LIN {X -0.056,Y -514.496,Z 256.006,A 0.000,B 0.000,C 90.000,E1 217.076} C_DIS
LIN {X -0.191,Y -508.629,Z 255.995,A 0.000,B 0.000,C 90.000,E1 215.025} C_DIS
LIN {X 0.078,Y -502.743,Z 255.983,A 0.000,B 0.000,C 90.000,E1 212.911} C_DIS
LIN {X -0.204,Y -496.416,Z 255.970,A 0.000,B 0.000,C 90.000,E1 210.541} C_DIS
LIN {X 0.173,Y -489.660,Z 255.954,A 0.000,B 0.000,C 90.000,E1 207.769} C_DIS
LIN {X -0.155,Y -484.810,Z 255.943,A 0.000,B 0.000,C 90.000,E1 205.668} C_DIS
LIN {X -0.161,Y -481.730,Z 255.934,A 0.000,B 0.000,C 90.000,E1 204.131} C_DIS
LIN {X -0.246,Y -475.770,Z 255.917,A 0.000,B 0.000,C 90.000,E1 201.046} C_DIS
LIN {X -0.152,Y -472.029,Z 255.905,A 0.000,B 0.000,C 90.000,E1 198.852} C_DIS
LIN {X -0.121,Y -469.175,Z 255.894,A 0.000,B 0.000,C 90.000,E1 196.968} C_DIS
LIN {X -0.013,Y -465.218,Z 255.878,A 0.000,B 0.000,C 90.000,E1 194.120} C_DIS
LIN {X -0.052,Y -462.080,Z 255.864,A 0.000,B 0.000,C 90.000,E1 191.591} C_DIS
LIN {X -0.160,Y -459.448,Z 255.852,A 0.000,B 0.000,C 90.000,E1 189.378} C_DIS
LIN {X 0.145,Y -456.317,Z 255.834,A 0.000,B 0.000,C 90.000,E1 186.144} C_DIS
LIN {X 0.227,Y -454.873,Z 255.825,A 0.000,B 0.000,C 90.000,E1 184.531} C_DIS
LIN {X -0.154,Y -452.914,Z 255.811,A 0.000,B 0.000,C 90.000,E1 182.007} C_DIS
LIN {X -0.154,Y -451.217,Z 255.797,A 0.000,B 0.000,C 90.000,E1 179.427} C_DIS
LIN {X 0.122,Y -449.780,Z 255.779,A 0.000,B 0.000,C 90.000,E1 176.159} C_DIS
LIN {X -0.156,Y -449.219,Z 255.763,A 0.000,B 0.000,C 90.000,E1 173.280} C_DIS
LIN {X 0.169,Y -449.233,Z 255.750,A 0.000,B 0.000,C 90.000,E1 170.971} C_DIS
LIN {X 0.184,Y -449.519,Z 255.737,A 0.000,B 0.000,C 90.000,E1 168.701} C_DIS
LIN {X -0.044,Y -450.253,Z 255.725,A 0.000,B 0.000,C 90.000,E1 166.464} C_DIS
LIN {X -0.134,Y -451.084,Z 255.712,A 0.000,B 0.000,C 90.000,E1 164.212} C_DIS
LIN {X 0.059,Y -453.464,Z 255.691,A 0.000,B 0.000,C 90.000,E1 160.315} C_DIS
LIN {X -0.251,Y -455.300,Z 255.678,A 0.000,B 0.000,C 90.000,E1 158.103} C_DIS
LIN {X 0.172,Y -457.927,Z 255.664,A 0.000,B 0.000,C 90.000,E1 155.485} C_DIS
LIN {X 0.008,Y -460.197,Z 255.653,A 0.000,B 0.000,C 90.000,E1 153.589} C_DIS
LIN {X -0.052,Y -463.628,Z 255.639,A 0.000,B 0.000,C 90.000,E1 151.051} C_DIS
LIN {X 0.071,Y -466.924,Z 255.627,A 0.000,B 0.000,C 90.000,E1 148.820} C_DIS
LIN {X -0.029,Y -470.471,Z 255.615,A 0.000,B 0.000,C 90.000,E1 146.628} C_DIS
LIN {X 0.014,Y -473.098,Z 255.606,A 0.000,B 0.000,C 90.000,E1 145.055} C_DIS
LIN {X 0.198,Y -475.136,Z 255.599,A 0.000,B 0.000,C 90.000,E1 143.783} C_DIS
LIN {X -0.172,Y -477.555,Z 255.590,A 0.000,B 0.000,C 90.000,E1 142.271} C_DIS
LIN {X -0.004,Y -479.372,Z 255.583,A 0.000,B 0.000,C 90.000,E1 141.009} C_DIS
LIN {X 0.002,Y -481.459,Z 255.575,A 0.000,B 0.000,C 90.000,E1 139.461} C_DIS
LIN {X 0.056,Y -482.599,Z 255.570,A 0.000,B 0.000,C 90.000,E1 138.528} C_DIS
LIN {X -0.199,Y -483.537,Z 255.565,A 0.000,B 0.000,C 90.000,E1 137.634} C_DIS
LIN {X -0.122,Y -484.313,Z 255.559,A 0.000,B 0.000,C 90.000,E1 136.701} C_DIS
LIN {X 0.157,Y -484.767,Z 255.556,A 0.000,B 0.000,C 90.000,E1 136.053} C_DIS
LIN {X -0.101,Y -485.206,Z 255.551,A 0.000,B 0.000,C 90.000,E1 135.162} C_DIS
LIN {X -0.208,Y -485.519,Z 255.544,A 0.000,B 0.000,C 90.000,E1 133.947} C_DIS
LIN {X 0.037,Y -485.533,Z 255.537,A 0.000,B 0.000,C 90.000,E1 132.690} C_DIS
LIN {X 0.139,Y -485.188,Z 255.532,A 0.000,B 0.000,C 90.000,E1 131.757} C_DIS
LIN {X -0.084,Y -484.586,Z 255.527,A 0.000,B 0.000,C 90.000,E1 130.862} C_DIS
LIN {X -0.054,Y -483.210,Z 255.518,A 0.000,B 0.000,C 90.000,E1 129.322} C_DIS
LIN {X -0.109,Y -481.993,Z 255.512,A 0.000,B 0.000,C 90.000,E1 128.096} C_DIS
LIN {X 0.011,Y -480.887,Z 255.506,A 0.000,B 0.000,C 90.000,E1 127.156} C_DIS
LIN {X -0.077,Y -479.167,Z 255.500,A 0.000,B 0.000,C 90.000,E1 125.931} C_DIS
LIN {X -0.081,Y -477.204,Z 255.493,A 0.000,B 0.000,C 90.000,E1 124.692} C_DIS
LIN {X -0.316,Y -474.649,Z 255.484,A 0.000,B 0.000,C 90.000,E1 123.166} C_DIS
LIN {X 0.192,Y -471.941,Z 255.475,A 0.000,B 0.000,C 90.000,E1 121.544} C_DIS
LIN {X -0.004,Y -469.141,Z 255.467,A 0.000,B 0.000,C 90.000,E1 120.001} C_DIS
LIN {X -0.078,Y -466.323,Z 255.458,A 0.000,B 0.000,C 90.000,E1 118.437} C_DIS
LIN {X -0.073,Y -462.933,Z 255.447,A 0.000,B 0.000,C 90.000,E1 116.539} C_DIS
LIN {X -0.154,Y -459.465,Z 255.437,A 0.000,B 0.000,C 90.000,E1 114.643} C_DIS
LIN {X -0.074,Y -456.086,Z 255.426,A 0.000,B 0.000,C 90.000,E1 112.717} C_DIS
LIN {X 0.041,Y -453.504,Z 255.418,A 0.000,B 0.000,C 90.000,E1 111.173} C_DIS
LIN {X 0.002,Y -453.518,Z 255.418,A 0.000,B 0.000,C 90.000,E1 111.173} C_DIS
LIN {X 0.044,Y -457.232,Z 255.410,A 0.000,B 0.000,C 90.000,E1 109.812} C_DIS
LIN {X 0.114,Y -465.853,Z 255.387,A 0.000,B 0.000,C 90.000,E1 105.662} C_DIS
LIN {X -0.166,Y -467.413,Z 255.384,A 0.000,B 0.000,C 90.000,E1 105.064} C_DIS
LIN {X 0.090,Y -468.042,Z 255.382,A 0.000,B 0.000,C 90.000,E1 104.717} C_DIS
LIN {X 0.230,Y -475.673,Z 255.357,A 0.000,B 0.000,C 90.000,E1 100.310} C_DIS
LIN {X 0.067,Y -476.249,Z 255.356,A 0.000,B 0.000,C 90.000,E1 100.018} C_DIS
LIN {X -0.148,Y -482.140,Z 255.330,A 0.000,B 0.000,C 90.000,E1 95.391} C_DIS
LIN {X 0.087,Y -485.533,Z 255.304,A 0.000,B 0.000,C 90.000,E1 90.745} C_DIS
LIN {X 0.119,Y -486.378,Z 255.280,A 0.000,B 0.000,C 90.000,E1 86.445} C_DIS
LIN {X -0.056,Y -486.344,Z 255.279,A 0.000,B 0.000,C 90.000,E1 86.159} C_DIS
LIN {X 0.022,Y -484.656,Z 255.253,A 0.000,B 0.000,C 90.000,E1 81.546} C_DIS
LIN {X -0.087,Y -480.577,Z 255.227,A 0.000,B 0.000,C 90.000,E1 76.937} C_DIS
LIN {X 0.060,Y -479.143,Z 255.222,A 0.000,B 0.000,C 90.000,E1 75.992} C_DIS
LIN {X 0.111,Y -473.974,Z 255.200,A 0.000,B 0.000,C 90.000,E1 71.945} C_DIS
LIN {X -0.018,Y -467.184,Z 255.179,A 0.000,B 0.000,C 90.000,E1 68.156} C_DIS
LIN {X -0.058,Y -467.189,Z 255.179,A 0.000,B 0.000,C 90.000,E1 68.156} C_DIS
LIN {X -0.001,Y -472.733,Z 255.167,A 0.000,B 0.000,C 90.000,E1 65.997} C_DIS
LIN {X -0.240,Y -477.581,Z 255.156,A 0.000,B 0.000,C 90.000,E1 64.152} C_DIS
LIN {X -0.147,Y -482.513,Z 255.146,A 0.000,B 0.000,C 90.000,E1 62.281} C_DIS
LIN {X 0.056,Y -487.565,Z 255.136,A 0.000,B 0.000,C 90.000,E1 60.411} C_DIS
LIN {X 0.179,Y -491.917,Z 255.127,A 0.000,B 0.000,C 90.000,E1 58.869} C_DIS
LIN {X -0.031,Y -496.228,Z 255.119,A 0.000,B 0.000,C 90.000,E1 57.375} C_DIS
LIN {X -0.032,Y -499.521,Z 255.112,A 0.000,B 0.000,C 90.000,E1 56.167} C_DIS
LIN {X -0.244,Y -503.454,Z 255.104,A 0.000,B 0.000,C 90.000,E1 54.689} C_DIS
LIN {X 0.023,Y -506.437,Z 255.097,A 0.000,B 0.000,C 90.000,E1 53.463} C_DIS
LIN {X -0.063,Y -509.805,Z 255.089,A 0.000,B 0.000,C 90.000,E1 51.984} C_DIS
LIN {X -0.016,Y -511.649,Z 255.084,A 0.000,B 0.000,C 90.000,E1 51.090} C_DIS
LIN {X 0.057,Y -513.380,Z 255.079,A 0.000,B 0.000,C 90.000,E1 50.194} C_DIS
LIN {X 0.070,Y -515.422,Z 255.072,A 0.000,B 0.000,C 90.000,E1 49.013} C_DIS
LIN {X -0.207,Y -516.733,Z 255.067,A 0.000,B 0.000,C 90.000,E1 48.162} C_DIS
LIN {X 0.262,Y -517.836,Z 255.063,A 0.000,B 0.000,C 90.000,E1 47.229} C_DIS
LIN {X 0.292,Y -519.039,Z 255.056,A 0.000,B 0.000,C 90.000,E1 46.053} C_DIS
LIN {X 0.047,Y -519.721,Z 255.051,A 0.000,B 0.000,C 90.000,E1 45.202} C_DIS
LIN {X -0.193,Y -520.236,Z 255.046,A 0.000,B 0.000,C 90.000,E1 44.352} C_DIS
LIN {X -0.128,Y -520.649,Z 255.040,A 0.000,B 0.000,C 90.000,E1 43.176} C_DIS
LIN {X -0.056,Y -520.877,Z 255.033,A 0.000,B 0.000,C 90.000,E1 42.000} C_DIS
LIN {X -0.274,Y -520.884,Z 255.028,A 0.000,B 0.000,C 90.000,E1 41.148} C_DIS
LIN {X 0.183,Y -520.520,Z 255.022,A 0.000,B 0.000,C 90.000,E1 39.930} C_DIS
LIN {X 0.023,Y -520.071,Z 255.017,A 0.000,B 0.000,C 90.000,E1 39.072} C_DIS
LIN {X 0.135,Y -519.308,Z 255.011,A 0.000,B 0.000,C 90.000,E1 37.890} C_DIS
LIN {X -0.084,Y -518.271,Z 255.004,A 0.000,B 0.000,C 90.000,E1 36.744} C_DIS
LIN {X -0.257,Y -517.276,Z 254.999,A 0.000,B 0.000,C 90.000,E1 35.884} C_DIS
LIN {X -0.087,Y -515.730,Z 254.993,A 0.000,B 0.000,C 90.000,E1 34.692} C_DIS
LIN {X 0.048,Y -513.278,Z 254.983,A 0.000,B 0.000,C 90.000,E1 32.911} C_DIS
LIN {X -0.219,Y -511.185,Z 254.975,A 0.000,B 0.000,C 90.000,E1 31.465} C_DIS
LIN {X -0.063,Y -507.987,Z 254.962,A 0.000,B 0.000,C 90.000,E1 29.077} C_DIS
LIN {X 0.249,Y -505.724,Z 254.952,A 0.000,B 0.000,C 90.000,E1 27.257} C_DIS
LIN {X 0.276,Y -503.544,Z 254.942,A 0.000,B 0.000,C 90.000,E1 25.463} C_DIS
LIN {X 0.036,Y -501.671,Z 254.932,A 0.000,B 0.000,C 90.000,E1 23.695} C_DIS
LIN {X -0.129,Y -500.469,Z 254.925,A 0.000,B 0.000,C 90.000,E1 22.514} C_DIS
LIN {X 0.219,Y -499.068,Z 254.917,A 0.000,B 0.000,C 90.000,E1 20.972} C_DIS
LIN {X -0.212,Y -497.454,Z 254.907,A 0.000,B 0.000,C 90.000,E1 19.214} C_DIS
LIN {X -0.099,Y -496.153,Z 254.898,A 0.000,B 0.000,C 90.000,E1 17.692} C_DIS
LIN {X 0.103,Y -494.522,Z 254.887,A 0.000,B 0.000,C 90.000,E1 15.552} C_DIS
LIN {X 0.265,Y -493.107,Z 254.875,A 0.000,B 0.000,C 90.000,E1 13.411} C_DIS
LIN {X 0.044,Y -491.834,Z 254.861,A 0.000,B 0.000,C 90.000,E1 11.007} C_DIS
LIN {X 0.196,Y -491.031,Z 254.849,A 0.000,B 0.000,C 90.000,E1 8.859} C_DIS
LIN {X -0.224,Y -490.606,Z 254.838,A 0.000,B 0.000,C 90.000,E1 6.777} C_DIS
LIN {X -0.034,Y -490.436,Z 254.822,A 0.000,B 0.000,C 90.000,E1 4.012} C_DIS
LIN {X -0.143,Y -490.702,Z 254.810,A 0.000,B 0.000,C 90.000,E1 1.892} C_DIS
LIN {X 0.186,Y -491.314,Z 254.799,A 0.000,B 0.000,C 90.000,E1 359.771} C_DIS
LIN {X 0.115,Y -492.573,Z 254.787,A 0.000,B 0.000,C 90.000,E1 357.650} C_DIS
LIN {X 0.098,Y -494.186,Z 254.775,A 0.000,B 0.000,C 90.000,E1 355.527} C_DIS
LIN {X -0.213,Y -499.228,Z 254.750,A 0.000,B 0.000,C 90.000,E1 351.027} C_DIS
LIN {X -0.167,Y -502.389,Z 254.740,A 0.000,B 0.000,C 90.000,E1 349.218} C_DIS
LIN {X -0.124,Y -509.727,Z 254.723,A 0.000,B 0.000,C 90.000,E1 346.228} C_DIS
LIN {X -0.195,Y -513.762,Z 254.715,A 0.000,B 0.000,C 90.000,E1 344.755} C_DIS
LIN {X -0.064,Y -517.741,Z 254.707,A 0.000,B 0.000,C 90.000,E1 343.268} C_DIS
LIN {X -0.267,Y -526.091,Z 254.691,A 0.000,B 0.000,C 90.000,E1 340.369} C_DIS
LIN {X 0.006,Y -533.634,Z 254.678,A 0.000,B 0.000,C 90.000,E1 338.028} C_DIS
LIN {X 0.057,Y -539.498,Z 254.668,A 0.000,B 0.000,C 90.000,E1 336.305} C_DIS
LIN {X -0.062,Y -544.456,Z 254.661,A 0.000,B 0.000,C 90.000,E1 334.897} C_DIS
LIN {X -0.078,Y -548.466,Z 254.654,A 0.000,B 0.000,C 90.000,E1 333.768} C_DIS
LIN {X -0.030,Y -553.742,Z 254.646,A 0.000,B 0.000,C 90.000,E1 332.359} C_DIS
LIN {X -0.115,Y -559.028,Z 254.639,A 0.000,B 0.000,C 90.000,E1 330.973} C_DIS
LIN {X -0.098,Y -564.055,Z 254.631,A 0.000,B 0.000,C 90.000,E1 329.587} C_DIS
LIN {X 0.000,Y -568.930,Z 254.623,A 0.000,B 0.000,C 90.000,E1 328.201} C_DIS
LIN {X 0.102,Y -576.974,Z 254.611,A 0.000,B 0.000,C 90.000,E1 326.008} C_DIS
LIN {X -0.239,Y -582.224,Z 254.604,A 0.000,B 0.000,C 90.000,E1 324.689} C_DIS
LIN {X -0.054,Y -585.203,Z 254.599,A 0.000,B 0.000,C 90.000,E1 323.863} C_DIS
LIN {X 0.234,Y -588.960,Z 254.593,A 0.000,B 0.000,C 90.000,E1 322.763} C_DIS
LIN {X -0.032,Y -593.351,Z 254.586,A 0.000,B 0.000,C 90.000,E1 321.457} C_DIS
LIN {X -0.234,Y -599.645,Z 254.576,A 0.000,B 0.000,C 90.000,E1 319.622} C_DIS
LIN {X -0.004,Y -604.266,Z 254.568,A 0.000,B 0.000,C 90.000,E1 318.286} C_DIS
LIN {X -0.016,Y -610.757,Z 254.558,A 0.000,B 0.000,C 90.000,E1 316.458} C_DIS
LIN {X 0.317,Y -613.455,Z 254.554,A 0.000,B 0.000,C 90.000,E1 315.648} C_DIS
LIN {X -0.353,Y -616.638,Z 254.548,A 0.000,B 0.000,C 90.000,E1 314.676} C_DIS
LIN {X 0.044,Y -618.801,Z 254.544,A 0.000,B 0.000,C 90.000,E1 313.866} C_DIS
LIN {X -0.114,Y -621.419,Z 254.538,A 0.000,B 0.000,C 90.000,E1 312.852} C_DIS
LIN {X -0.237,Y -623.831,Z 254.532,A 0.000,B 0.000,C 90.000,E1 311.838} C_DIS
LIN {X 0.141,Y -625.862,Z 254.527,A 0.000,B 0.000,C 90.000,E1 310.782} C_DIS
LIN {X 0.011,Y -628.124,Z 254.520,A 0.000,B 0.000,C 90.000,E1 309.519} C_DIS
LIN {X -0.046,Y -629.602,Z 254.514,A 0.000,B 0.000,C 90.000,E1 308.508} C_DIS
LIN {X -0.382,Y -630.898,Z 254.508,A 0.000,B 0.000,C 90.000,E1 307.523} C_DIS
LIN {X -0.172,Y -631.687,Z 254.504,A 0.000,B 0.000,C 90.000,E1 306.744} C_DIS
LIN {X 0.050,Y -632.244,Z 254.500,A 0.000,B 0.000,C 90.000,E1 305.964} C_DIS
LIN {X -0.239,Y -632.585,Z 254.496,A 0.000,B 0.000,C 90.000,E1 305.231} C_DIS
LIN {X -0.151,Y -632.800,Z 254.487,A 0.000,B 0.000,C 90.000,E1 303.706} C_DIS
LIN {X -0.278,Y -632.632,Z 254.483,A 0.000,B 0.000,C 90.000,E1 302.959} C_DIS
LIN {X -0.405,Y -632.178,Z 254.479,A 0.000,B 0.000,C 90.000,E1 302.212} C_DIS
LIN {X 0.001,Y -631.406,Z 254.475,A 0.000,B 0.000,C 90.000,E1 301.416} C_DIS
LIN {X -0.139,Y -630.389,Z 254.470,A 0.000,B 0.000,C 90.000,E1 300.669} C_DIS
LIN {X 0.250,Y -629.069,Z 254.466,A 0.000,B 0.000,C 90.000,E1 299.873} C_DIS
LIN {X 0.091,Y -627.074,Z 254.460,A 0.000,B 0.000,C 90.000,E1 298.871} C_DIS
LIN {X 0.153,Y -624.685,Z 254.455,A 0.000,B 0.000,C 90.000,E1 297.847} C_DIS
LIN {X 0.191,Y -622.134,Z 254.449,A 0.000,B 0.000,C 90.000,E1 296.821} C_DIS
LIN {X 0.183,Y -618.018,Z 254.441,A 0.000,B 0.000,C 90.000,E1 295.283} C_DIS
LIN {X 0.021,Y -611.228,Z 254.426,A 0.000,B 0.000,C 90.000,E1 292.717} C_DIS
LIN {X 0.303,Y -606.098,Z 254.415,A 0.000,B 0.000,C 90.000,E1 290.610} C_DIS
LIN {X 0.296,Y -601.870,Z 254.405,A 0.000,B 0.000,C 90.000,E1 288.779} C_DIS
LIN {X 0.133,Y -595.753,Z 254.388,A 0.000,B 0.000,C 90.000,E1 285.898} C_DIS
LIN {X 0.163,Y -590.972,Z 254.374,A 0.000,B 0.000,C 90.000,E1 283.244} C_DIS
LIN {X 0.164,Y -586.780,Z 254.357,A 0.000,B 0.000,C 90.000,E1 280.310} C_DIS
LIN {X -0.029,Y -584.653,Z 254.347,A 0.000,B 0.000,C 90.000,E1 278.454} C_DIS
LIN {X 0.236,Y -583.017,Z 254.337,A 0.000,B 0.000,C 90.000,E1 276.549} C_DIS
LIN {X -0.166,Y -581.377,Z 254.322,A 0.000,B 0.000,C 90.000,E1 273.898} C_DIS
LIN {X -0.207,Y -581.187,Z 254.292,A 0.000,B 0.000,C 90.000,E1 268.511} C_DIS
LIN {X -0.180,Y -583.405,Z 254.272,A 0.000,B 0.000,C 90.000,E1 265.008} C_DIS
LIN {X 0.248,Y -585.602,Z 254.260,A 0.000,B 0.000,C 90.000,E1 262.818} C_DIS
LIN {X -0.028,Y -587.943,Z 254.250,A 0.000,B 0.000,C 90.000,E1 260.971} C_DIS
LIN {X -0.111,Y -591.502,Z 254.237,A 0.000,B 0.000,C 90.000,E1 258.578} C_DIS
LIN {X -0.209,Y -593.947,Z 254.228,A 0.000,B 0.000,C 90.000,E1 256.992} C_DIS
LIN {X -0.265,Y -596.421,Z 254.219,A 0.000,B 0.000,C 90.000,E1 255.408} C_DIS
LIN {X 0.161,Y -597.600,Z 254.214,A 0.000,B 0.000,C 90.000,E1 254.574} C_DIS
LIN {X -0.259,Y -598.967,Z 254.209,A 0.000,B 0.000,C 90.000,E1 253.559} C_DIS
LIN {X 0.196,Y -599.745,Z 254.204,A 0.000,B 0.000,C 90.000,E1 252.725} C_DIS
LIN {X 0.085,Y -600.305,Z 254.200,A 0.000,B 0.000,C 90.000,E1 251.945} C_DIS
LIN {X -0.119,Y -600.723,Z 254.194,A 0.000,B 0.000,C 90.000,E1 250.913} C_DIS
LIN {X -0.315,Y -600.910,Z 254.188,A 0.000,B 0.000,C 90.000,E1 249.880} C_DIS
LIN {X -0.217,Y -600.859,Z 254.184,A 0.000,B 0.000,C 90.000,E1 249.082} C_DIS
LIN {X -0.117,Y -600.439,Z 254.179,A 0.000,B 0.000,C 90.000,E1 248.284} C_DIS
LIN {X -0.026,Y -599.780,Z 254.175,A 0.000,B 0.000,C 90.000,E1 247.486} C_DIS
LIN {X 0.290,Y -598.927,Z 254.171,A 0.000,B 0.000,C 90.000,E1 246.666} C_DIS
LIN {X -0.188,Y -597.871,Z 254.166,A 0.000,B 0.000,C 90.000,E1 245.921} C_DIS
LIN {X 0.112,Y -596.519,Z 254.162,A 0.000,B 0.000,C 90.000,E1 245.101} C_DIS
LIN {X 0.307,Y -594.341,Z 254.156,A 0.000,B 0.000,C 90.000,E1 244.024} C_DIS
LIN {X 0.033,Y -592.542,Z 254.151,A 0.000,B 0.000,C 90.000,E1 243.256} C_DIS
LIN {X 0.334,Y -589.273,Z 254.144,A 0.000,B 0.000,C 90.000,E1 241.897} C_DIS
LIN {X 0.004,Y -587.228,Z 254.140,A 0.000,B 0.000,C 90.000,E1 241.129} C_DIS
LIN {X -0.062,Y -585.062,Z 254.135,A 0.000,B 0.000,C 90.000,E1 240.333} C_DIS
LIN {X -0.149,Y -582.754,Z 254.131,A 0.000,B 0.000,C 90.000,E1 239.537} C_DIS
LIN {X -0.260,Y -580.298,Z 254.126,A 0.000,B 0.000,C 90.000,E1 238.742} C_DIS
LIN {X -0.259,Y -575.026,Z 254.117,A 0.000,B 0.000,C 90.000,E1 237.120} C_DIS
LIN {X 0.197,Y -568.008,Z 254.105,A 0.000,B 0.000,C 90.000,E1 234.895} C_DIS
LIN {X 0.116,Y -562.908,Z 254.096,A 0.000,B 0.000,C 90.000,E1 233.256} C_DIS
LIN {X -0.076,Y -557.777,Z 254.087,A 0.000,B 0.000,C 90.000,E1 231.618} C_DIS
LIN {X -0.113,Y -553.502,Z 254.079,A 0.000,B 0.000,C 90.000,E1 230.231} C_DIS
LIN {X -0.293,Y -549.165,Z 254.071,A 0.000,B 0.000,C 90.000,E1 228.852} C_DIS
LIN {X -0.171,Y -545.655,Z 254.065,A 0.000,B 0.000,C 90.000,E1 227.715} C_DIS
LIN {X -0.119,Y -541.133,Z 254.057,A 0.000,B 0.000,C 90.000,E1 226.296} C_DIS
LIN {X -0.140,Y -537.527,Z 254.051,A 0.000,B 0.000,C 90.000,E1 225.162} C_DIS
LIN {X -0.210,Y -533.902,Z 254.045,A 0.000,B 0.000,C 90.000,E1 224.028} C_DIS
LIN {X -0.066,Y -527.628,Z 254.033,A 0.000,B 0.000,C 90.000,E1 222.000} C_DIS
LIN {X -0.034,Y -521.418,Z 254.022,A 0.000,B 0.000,C 90.000,E1 219.967} C_DIS
LIN {X -0.170,Y -515.355,Z 254.011,A 0.000,B 0.000,C 90.000,E1 217.935} C_DIS
LIN {X -0.119,Y -511.111,Z 254.003,A 0.000,B 0.000,C 90.000,E1 216.457} C_DIS
LIN {X 0.155,Y -506.916,Z 253.994,A 0.000,B 0.000,C 90.000,E1 214.945} C_DIS
LIN {X -0.051,Y -501.042,Z 253.983,A 0.000,B 0.000,C 90.000,E1 212.880} C_DIS
LIN {X -0.247,Y -495.472,Z 253.971,A 0.000,B 0.000,C 90.000,E1 210.797} C_DIS
LIN {X 0.009,Y -490.835,Z 253.961,A 0.000,B 0.000,C 90.000,E1 208.949} C_DIS
LIN {X -0.067,Y -485.834,Z 253.949,A 0.000,B 0.000,C 90.000,E1 206.821} C_DIS
LIN {X 0.152,Y -480.021,Z 253.934,A 0.000,B 0.000,C 90.000,E1 204.027} C_DIS
LIN {X 0.189,Y -474.119,Z 253.916,A 0.000,B 0.000,C 90.000,E1 200.918} C_DIS
LIN {X -0.009,Y -469.450,Z 253.901,A 0.000,B 0.000,C 90.000,E1 198.127} C_DIS
LIN {X -0.179,Y -466.632,Z 253.890,A 0.000,B 0.000,C 90.000,E1 196.260} C_DIS
LIN {X 0.146,Y -463.648,Z 253.878,A 0.000,B 0.000,C 90.000,E1 194.008} C_DIS
LIN {X -0.175,Y -460.914,Z 253.866,A 0.000,B 0.000,C 90.000,E1 191.827} C_DIS
LIN {X -0.077,Y -457.902,Z 253.851,A 0.000,B 0.000,C 90.000,E1 189.265} C_DIS
LIN {X 0.010,Y -455.059,Z 253.835,A 0.000,B 0.000,C 90.000,E1 186.372} C_DIS
LIN {X -0.224,Y -453.357,Z 253.825,A 0.000,B 0.000,C 90.000,E1 184.473} C_DIS
LIN {X -0.196,Y -451.380,Z 253.810,A 0.000,B 0.000,C 90.000,E1 181.892} C_DIS
LIN {X 0.048,Y -449.892,Z 253.798,A 0.000,B 0.000,C 90.000,E1 179.599} C_DIS
LIN {X -0.174,Y -448.418,Z 253.780,A 0.000,B 0.000,C 90.000,E1 176.388} C_DIS
LIN {X -0.046,Y -447.827,Z 253.764,A 0.000,B 0.000,C 90.000,E1 173.451} C_DIS
LIN {X -0.008,Y -447.816,Z 253.749,A 0.000,B 0.000,C 90.000,E1 170.849} C_DIS
LIN {X 0.233,Y -448.098,Z 253.738,A 0.000,B 0.000,C 90.000,E1 168.870} C_DIS
LIN {X 0.056,Y -448.949,Z 253.724,A 0.000,B 0.000,C 90.000,E1 166.297} C_DIS
LIN {X 0.042,Y -449.838,Z 253.711,A 0.000,B 0.000,C 90.000,E1 164.031} C_DIS
LIN {X -0.179,Y -451.530,Z 253.695,A 0.000,B 0.000,C 90.000,E1 161.148} C_DIS
LIN {X 0.049,Y -453.599,Z 253.681,A 0.000,B 0.000,C 90.000,E1 158.539} C_DIS
LIN {X -0.001,Y -456.086,Z 253.667,A 0.000,B 0.000,C 90.000,E1 155.973} C_DIS
LIN {X 0.120,Y -458.710,Z 253.654,A 0.000,B 0.000,C 90.000,E1 153.717} C_DIS
LIN {X 0.144,Y -462.606,Z 253.638,A 0.000,B 0.000,C 90.000,E1 150.845} C_DIS
LIN {X 0.100,Y -465.443,Z 253.628,A 0.000,B 0.000,C 90.000,E1 148.948} C_DIS
LIN {X -0.037,Y -468.964,Z 253.615,A 0.000,B 0.000,C 90.000,E1 146.755} C_DIS
LIN {X -0.242,Y -472.132,Z 253.605,A 0.000,B 0.000,C 90.000,E1 144.895} C_DIS
LIN {X 0.097,Y -474.616,Z 253.596,A 0.000,B 0.000,C 90.000,E1 143.290} C_DIS
LIN {X 0.009,Y -477.006,Z 253.588,A 0.000,B 0.000,C 90.000,E1 141.743} C_DIS
LIN {X -0.026,Y -479.152,Z 253.579,A 0.000,B 0.000,C 90.000,E1 140.194} C_DIS
LIN {X -0.031,Y -481.112,Z 253.570,A 0.000,B 0.000,C 90.000,E1 138.647} C_DIS
LIN {X 0.143,Y -482.357,Z 253.563,A 0.000,B 0.000,C 90.000,E1 137.391} C_DIS
LIN {X -0.006,Y -483.277,Z 253.557,A 0.000,B 0.000,C 90.000,E1 136.176} C_DIS
LIN {X 0.207,Y -483.877,Z 253.550,A 0.000,B 0.000,C 90.000,E1 134.919} C_DIS
LIN {X 0.080,Y -484.157,Z 253.543,A 0.000,B 0.000,C 90.000,E1 133.704} C_DIS
LIN {X -0.024,Y -484.103,Z 253.536,A 0.000,B 0.000,C 90.000,E1 132.486} C_DIS
LIN {X 0.065,Y -483.687,Z 253.531,A 0.000,B 0.000,C 90.000,E1 131.553} C_DIS
LIN {X 0.144,Y -483.046,Z 253.526,A 0.000,B 0.000,C 90.000,E1 130.620} C_DIS
LIN {X 0.021,Y -481.978,Z 253.519,A 0.000,B 0.000,C 90.000,E1 129.402} C_DIS
LIN {X -0.051,Y -480.771,Z 253.512,A 0.000,B 0.000,C 90.000,E1 128.177} C_DIS
LIN {X -0.135,Y -479.324,Z 253.505,A 0.000,B 0.000,C 90.000,E1 126.950} C_DIS
LIN {X 0.144,Y -477.589,Z 253.498,A 0.000,B 0.000,C 90.000,E1 125.678} C_DIS
LIN {X 0.185,Y -475.135,Z 253.490,A 0.000,B 0.000,C 90.000,E1 124.119} C_DIS
LIN {X -0.058,Y -473.600,Z 253.485,A 0.000,B 0.000,C 90.000,E1 123.214} C_DIS
LIN {X -0.227,Y -470.913,Z 253.476,A 0.000,B 0.000,C 90.000,E1 121.671} C_DIS
LIN {X 0.124,Y -467.564,Z 253.465,A 0.000,B 0.000,C 90.000,E1 119.745} C_DIS
LIN {X 0.022,Y -464.762,Z 253.457,A 0.000,B 0.000,C 90.000,E1 118.180} C_DIS
LIN {X -0.010,Y -461.341,Z 253.446,A 0.000,B 0.000,C 90.000,E1 116.283} C_DIS
LIN {X -0.039,Y -458.462,Z 253.437,A 0.000,B 0.000,C 90.000,E1 114.695} C_DIS
LIN {X 0.010,Y -455.098,Z 253.427,A 0.000,B 0.000,C 90.000,E1 112.770} C_DIS
LIN {X -0.161,Y -452.838,Z 253.419,A 0.000,B 0.000,C 90.000,E1 111.461} C_DIS
LIN {X 0.222,Y -452.834,Z 253.419,A 0.000,B 0.000,C 90.000,E1 111.408} C_DIS
LIN {X -0.058,Y -457.072,Z 253.410,A 0.000,B 0.000,C 90.000,E1 109.885} C_DIS
LIN {X 0.113,Y -460.774,Z 253.400,A 0.000,B 0.000,C 90.000,E1 107.946} C_DIS
LIN {X -0.253,Y -467.264,Z 253.384,A 0.000,B 0.000,C 90.000,E1 105.134} C_DIS
LIN {X 0.123,Y -467.959,Z 253.382,A 0.000,B 0.000,C 90.000,E1 104.773} C_DIS
LIN {X 0.087,Y -476.178,Z 253.356,A 0.000,B 0.000,C 90.000,E1 100.074} C_DIS
LIN {X -0.137,Y -482.084,Z 253.330,A 0.000,B 0.000,C 90.000,E1 95.448} C_DIS
LIN {X 0.092,Y -485.503,Z 253.305,A 0.000,B 0.000,C 90.000,E1 90.802} C_DIS
LIN {X 0.125,Y -486.383,Z 253.281,A 0.000,B 0.000,C 90.000,E1 86.502} C_DIS
LIN {X -0.051,Y -486.361,Z 253.279,A 0.000,B 0.000,C 90.000,E1 86.216} C_DIS
LIN {X 0.032,Y -484.685,Z 253.253,A 0.000,B 0.000,C 90.000,E1 81.602} C_DIS
LIN {X -0.067,Y -480.608,Z 253.228,A 0.000,B 0.000,C 90.000,E1 76.992} C_DIS
LIN {X -0.209,Y -480.248,Z 253.226,A 0.000,B 0.000,C 90.000,E1 76.700} C_DIS
LIN {X 0.147,Y -474.077,Z 253.200,A 0.000,B 0.000,C 90.000,E1 72.000} C_DIS
LIN {X -0.140,Y -466.789,Z 253.177,A 0.000,B 0.000,C 90.000,E1 67.901} C_DIS
LIN {X 0.252,Y -466.788,Z 253.177,A 0.000,B 0.000,C 90.000,E1 67.847} C_DIS
LIN {X 0.035,Y -471.482,Z 253.167,A 0.000,B 0.000,C 90.000,E1 66.049} C_DIS
LIN {X 0.204,Y -476.346,Z 253.157,A 0.000,B 0.000,C 90.000,E1 64.152} C_DIS
LIN {X 0.049,Y -481.256,Z 253.146,A 0.000,B 0.000,C 90.000,E1 62.308} C_DIS
LIN {X 0.257,Y -487.144,Z 253.134,A 0.000,B 0.000,C 90.000,E1 60.127} C_DIS
LIN {X 0.125,Y -491.450,Z 253.126,A 0.000,B 0.000,C 90.000,E1 58.614} C_DIS
LIN {X -0.098,Y -495.748,Z 253.117,A 0.000,B 0.000,C 90.000,E1 57.120} C_DIS
LIN {X 0.166,Y -499.004,Z 253.111,A 0.000,B 0.000,C 90.000,E1 55.881} C_DIS
LIN {X -0.051,Y -502.860,Z 253.102,A 0.000,B 0.000,C 90.000,E1 54.402} C_DIS
LIN {X -0.094,Y -505.760,Z 253.096,A 0.000,B 0.000,C 90.000,E1 53.210} C_DIS
LIN {X 0.207,Y -508.449,Z 253.089,A 0.000,B 0.000,C 90.000,E1 51.984} C_DIS
LIN {X 0.240,Y -510.291,Z 253.084,A 0.000,B 0.000,C 90.000,E1 51.090} C_DIS
LIN {X 0.212,Y -512.523,Z 253.077,A 0.000,B 0.000,C 90.000,E1 49.908} C_DIS
LIN {X -0.178,Y -514.498,Z 253.071,A 0.000,B 0.000,C 90.000,E1 48.771} C_DIS
LIN {X 0.184,Y -516.097,Z 253.064,A 0.000,B 0.000,C 90.000,E1 47.553} C_DIS
LIN {X 0.188,Y -517.358,Z 253.058,A 0.000,B 0.000,C 90.000,E1 46.377} C_DIS
LIN {X -0.164,Y -518.308,Z 253.051,A 0.000,B 0.000,C 90.000,E1 45.243} C_DIS
LIN {X 0.232,Y -518.951,Z 253.045,A 0.000,B 0.000,C 90.000,E1 44.028} C_DIS
LIN {X 0.277,Y -519.316,Z 253.038,A 0.000,B 0.000,C 90.000,E1 42.852} C_DIS
LIN {X 0.044,Y -519.461,Z 253.033,A 0.000,B 0.000,C 90.000,E1 42.000} C_DIS
LIN {X -0.188,Y -519.437,Z 253.029,A 0.000,B 0.000,C 90.000,E1 41.148} C_DIS
LIN {X -0.030,Y -519.196,Z 253.024,A 0.000,B 0.000,C 90.000,E1 40.253} C_DIS
LIN {X 0.071,Y -518.638,Z 253.017,A 0.000,B 0.000,C 90.000,E1 39.072} C_DIS
LIN {X 0.161,Y -517.880,Z 253.011,A 0.000,B 0.000,C 90.000,E1 37.890} C_DIS
LIN {X -0.077,Y -516.773,Z 253.004,A 0.000,B 0.000,C 90.000,E1 36.744} C_DIS
LIN {X 0.035,Y -515.742,Z 252.999,A 0.000,B 0.000,C 90.000,E1 35.851} C_DIS
LIN {X -0.121,Y -514.162,Z 252.993,A 0.000,B 0.000,C 90.000,E1 34.692} C_DIS
LIN {X 0.257,Y -511.613,Z 252.983,A 0.000,B 0.000,C 90.000,E1 32.880} C_DIS
LIN {X 0.117,Y -509.467,Z 252.975,A 0.000,B 0.000,C 90.000,E1 31.416} C_DIS
LIN {X -0.212,Y -506.201,Z 252.961,A 0.000,B 0.000,C 90.000,E1 29.077} C_DIS
LIN {X 0.135,Y -503.552,Z 252.950,A 0.000,B 0.000,C 90.000,E1 26.950} C_DIS
LIN {X 0.048,Y -501.793,Z 252.942,A 0.000,B 0.000,C 90.000,E1 25.463} C_DIS
LIN {X 0.228,Y -499.900,Z 252.932,A 0.000,B 0.000,C 90.000,E1 23.643} C_DIS
LIN {X 0.040,Y -498.707,Z 252.925,A 0.000,B 0.000,C 90.000,E1 22.461} C_DIS
LIN {X -0.046,Y -497.023,Z 252.915,A 0.000,B 0.000,C 90.000,E1 20.663} C_DIS
LIN {X -0.053,Y -495.429,Z 252.905,A 0.000,B 0.000,C 90.000,E1 18.852} C_DIS
LIN {X -0.021,Y -494.415,Z 252.898,A 0.000,B 0.000,C 90.000,E1 17.638} C_DIS
LIN {X 0.272,Y -492.783,Z 252.886,A 0.000,B 0.000,C 90.000,E1 15.481} C_DIS
LIN {X -0.219,Y -491.347,Z 252.874,A 0.000,B 0.000,C 90.000,E1 13.411} C_DIS
LIN {X 0.100,Y -490.215,Z 252.863,A 0.000,B 0.000,C 90.000,E1 11.243} C_DIS
LIN {X 0.101,Y -489.306,Z 252.849,A 0.000,B 0.000,C 90.000,E1 8.803} C_DIS
LIN {X 0.002,Y -488.781,Z 252.835,A 0.000,B 0.000,C 90.000,E1 6.372} C_DIS
LIN {X -0.229,Y -488.635,Z 252.822,A 0.000,B 0.000,C 90.000,E1 3.955} C_DIS
LIN {X 0.119,Y -488.933,Z 252.810,A 0.000,B 0.000,C 90.000,E1 1.776} C_DIS
LIN {X 0.026,Y -489.632,Z 252.797,A 0.000,B 0.000,C 90.000,E1 359.484} C_DIS
LIN {X 0.066,Y -490.729,Z 252.787,A 0.000,B 0.000,C 90.000,E1 357.650} C_DIS
LIN {X -0.158,Y -492.596,Z 252.774,A 0.000,B 0.000,C 90.000,E1 355.241} C_DIS
LIN {X 0.076,Y -497.330,Z 252.750,A 0.000,B 0.000,C 90.000,E1 350.971} C_DIS
LIN {X 0.078,Y -500.523,Z 252.740,A 0.000,B 0.000,C 90.000,E1 349.162} C_DIS
LIN {X 0.031,Y -510.386,Z 252.718,A 0.000,B 0.000,C 90.000,E1 345.283} C_DIS
LIN {X 0.108,Y -514.418,Z 252.710,A 0.000,B 0.000,C 90.000,E1 343.795} C_DIS
LIN {X 0.150,Y -521.748,Z 252.695,A 0.000,B 0.000,C 90.000,E1 341.148} C_DIS
LIN {X -0.207,Y -530.944,Z 252.679,A 0.000,B 0.000,C 90.000,E1 338.284} C_DIS
LIN {X -0.005,Y -536.820,Z 252.670,A 0.000,B 0.000,C 90.000,E1 336.538} C_DIS
LIN {X 0.098,Y -541.812,Z 252.662,A 0.000,B 0.000,C 90.000,E1 335.101} C_DIS
LIN {X -0.214,Y -549.976,Z 252.649,A 0.000,B 0.000,C 90.000,E1 332.871} C_DIS
LIN {X -0.102,Y -556.327,Z 252.640,A 0.000,B 0.000,C 90.000,E1 331.179} C_DIS
LIN {X -0.208,Y -560.463,Z 252.634,A 0.000,B 0.000,C 90.000,E1 330.078} C_DIS
LIN {X 0.111,Y -565.426,Z 252.626,A 0.000,B 0.000,C 90.000,E1 328.663} C_DIS
LIN {X -0.012,Y -572.334,Z 252.615,A 0.000,B 0.000,C 90.000,E1 326.755} C_DIS
LIN {X 0.202,Y -578.575,Z 252.606,A 0.000,B 0.000,C 90.000,E1 325.102} C_DIS
LIN {X 0.053,Y -582.706,Z 252.600,A 0.000,B 0.000,C 90.000,E1 324.036} C_DIS
LIN {X -0.037,Y -586.522,Z 252.594,A 0.000,B 0.000,C 90.000,E1 322.970} C_DIS
LIN {X -0.082,Y -590.078,Z 252.588,A 0.000,B 0.000,C 90.000,E1 321.904} C_DIS
LIN {X 0.020,Y -596.341,Z 252.578,A 0.000,B 0.000,C 90.000,E1 320.033} C_DIS
LIN {X 0.043,Y -601.973,Z 252.569,A 0.000,B 0.000,C 90.000,E1 318.447} C_DIS
LIN {X 0.168,Y -607.601,Z 252.560,A 0.000,B 0.000,C 90.000,E1 316.863} C_DIS
LIN {X 0.283,Y -611.292,Z 252.555,A 0.000,B 0.000,C 90.000,E1 315.810} C_DIS
LIN {X -0.243,Y -613.828,Z 252.550,A 0.000,B 0.000,C 90.000,E1 315.081} C_DIS
LIN {X 0.125,Y -616.143,Z 252.546,A 0.000,B 0.000,C 90.000,E1 314.271} C_DIS
LIN {X -0.066,Y -618.855,Z 252.540,A 0.000,B 0.000,C 90.000,E1 313.257} C_DIS
LIN {X 0.350,Y -620.735,Z 252.536,A 0.000,B 0.000,C 90.000,E1 312.447} C_DIS
LIN {X 0.363,Y -622.441,Z 252.532,A 0.000,B 0.000,C 90.000,E1 311.676} C_DIS
LIN {X -0.161,Y -624.436,Z 252.526,A 0.000,B 0.000,C 90.000,E1 310.701} C_DIS
LIN {X 0.224,Y -626.201,Z 252.520,A 0.000,B 0.000,C 90.000,E1 309.644} C_DIS
LIN {X 0.029,Y -627.049,Z 252.518,A 0.000,B 0.000,C 90.000,E1 309.152} C_DIS
LIN {X -0.049,Y -628.410,Z 252.512,A 0.000,B 0.000,C 90.000,E1 308.141} C_DIS
LIN {X 0.128,Y -629.325,Z 252.508,A 0.000,B 0.000,C 90.000,E1 307.363} C_DIS
LIN {X -0.039,Y -629.901,Z 252.505,A 0.000,B 0.000,C 90.000,E1 306.870} C_DIS
LIN {X 0.161,Y -630.473,Z 252.501,A 0.000,B 0.000,C 90.000,E1 306.091} C_DIS
LIN {X -0.151,Y -630.862,Z 252.495,A 0.000,B 0.000,C 90.000,E1 305.105} C_DIS
LIN {X -0.101,Y -631.054,Z 252.488,A 0.000,B 0.000,C 90.000,E1 303.833} C_DIS
LIN {X -0.248,Y -630.957,Z 252.484,A 0.000,B 0.000,C 90.000,E1 303.086} C_DIS
LIN {X 0.139,Y -630.531,Z 252.480,A 0.000,B 0.000,C 90.000,E1 302.291} C_DIS
LIN {X -0.026,Y -630.076,Z 252.477,A 0.000,B 0.000,C 90.000,E1 301.799} C_DIS
LIN {X -0.181,Y -629.116,Z 252.472,A 0.000,B 0.000,C 90.000,E1 301.052} C_DIS
LIN {X 0.190,Y -628.019,Z 252.468,A 0.000,B 0.000,C 90.000,E1 300.256} C_DIS
LIN {X 0.028,Y -625.572,Z 252.461,A 0.000,B 0.000,C 90.000,E1 298.999} C_DIS
LIN {X 0.060,Y -623.872,Z 252.457,A 0.000,B 0.000,C 90.000,E1 298.231} C_DIS
LIN {X 0.086,Y -620.711,Z 252.450,A 0.000,B 0.000,C 90.000,E1 296.950} C_DIS
LIN {X 0.064,Y -617.326,Z 252.443,A 0.000,B 0.000,C 90.000,E1 295.668} C_DIS
LIN {X 0.083,Y -609.800,Z 252.427,A 0.000,B 0.000,C 90.000,E1 292.823} C_DIS
LIN {X 0.096,Y -604.678,Z 252.415,A 0.000,B 0.000,C 90.000,E1 290.737} C_DIS
LIN {X 0.061,Y -600.455,Z 252.405,A 0.000,B 0.000,C 90.000,E1 288.906} C_DIS
LIN {X -0.142,Y -594.304,Z 252.389,A 0.000,B 0.000,C 90.000,E1 286.024} C_DIS
LIN {X 0.298,Y -589.930,Z 252.376,A 0.000,B 0.000,C 90.000,E1 283.592} C_DIS
LIN {X 0.001,Y -585.954,Z 252.361,A 0.000,B 0.000,C 90.000,E1 280.950} C_DIS
LIN {X 0.265,Y -583.143,Z 252.347,A 0.000,B 0.000,C 90.000,E1 278.511} C_DIS
LIN {X -0.072,Y -580.880,Z 252.333,A 0.000,B 0.000,C 90.000,E1 275.853} C_DIS
LIN {X -0.287,Y -579.302,Z 252.315,A 0.000,B 0.000,C 90.000,E1 272.636} C_DIS
LIN {X 0.223,Y -579.741,Z 252.289,A 0.000,B 0.000,C 90.000,E1 267.993} C_DIS
LIN {X 0.198,Y -581.551,Z 252.274,A 0.000,B 0.000,C 90.000,E1 265.298} C_DIS
LIN {X -0.177,Y -583.368,Z 252.264,A 0.000,B 0.000,C 90.000,E1 263.451} C_DIS
LIN {X 0.083,Y -585.604,Z 252.253,A 0.000,B 0.000,C 90.000,E1 261.546} C_DIS
LIN {X -0.104,Y -588.220,Z 252.243,A 0.000,B 0.000,C 90.000,E1 259.690} C_DIS
LIN {X -0.009,Y -591.103,Z 252.232,A 0.000,B 0.000,C 90.000,E1 257.813} C_DIS
LIN {X 0.189,Y -593.162,Z 252.225,A 0.000,B 0.000,C 90.000,E1 256.464} C_DIS
LIN {X -0.166,Y -595.213,Z 252.218,A 0.000,B 0.000,C 90.000,E1 255.172} C_DIS
LIN {X 0.248,Y -596.325,Z 252.213,A 0.000,B 0.000,C 90.000,E1 254.338} C_DIS
LIN {X -0.191,Y -597.641,Z 252.207,A 0.000,B 0.000,C 90.000,E1 253.323} C_DIS
LIN {X -0.322,Y -598.368,Z 252.203,A 0.000,B 0.000,C 90.000,E1 252.543} C_DIS
LIN {X 0.122,Y -598.872,Z 252.199,A 0.000,B 0.000,C 90.000,E1 251.710} C_DIS
LIN {X -0.105,Y -599.193,Z 252.193,A 0.000,B 0.000,C 90.000,E1 250.678} C_DIS
LIN {X -0.119,Y -599.324,Z 252.187,A 0.000,B 0.000,C 90.000,E1 249.625} C_DIS
LIN {X 0.054,Y -599.286,Z 252.184,A 0.000,B 0.000,C 90.000,E1 249.082} C_DIS
LIN {X 0.137,Y -598.907,Z 252.179,A 0.000,B 0.000,C 90.000,E1 248.284} C_DIS
LIN {X 0.212,Y -598.274,Z 252.175,A 0.000,B 0.000,C 90.000,E1 247.486} C_DIS
LIN {X 0.189,Y -597.069,Z 252.169,A 0.000,B 0.000,C 90.000,E1 246.433} C_DIS
LIN {X -0.067,Y -595.932,Z 252.165,A 0.000,B 0.000,C 90.000,E1 245.665} C_DIS
LIN {X 0.214,Y -594.485,Z 252.160,A 0.000,B 0.000,C 90.000,E1 244.845} C_DIS
LIN {X -0.151,Y -592.267,Z 252.155,A 0.000,B 0.000,C 90.000,E1 243.819} C_DIS
LIN {X 0.087,Y -590.407,Z 252.150,A 0.000,B 0.000,C 90.000,E1 242.999} C_DIS
LIN {X -0.170,Y -587.082,Z 252.143,A 0.000,B 0.000,C 90.000,E1 241.691} C_DIS
LIN {X 0.157,Y -584.294,Z 252.137,A 0.000,B 0.000,C 90.000,E1 240.589} C_DIS
LIN {X -0.071,Y -581.218,Z 252.131,A 0.000,B 0.000,C 90.000,E1 239.537} C_DIS
LIN {X -0.044,Y -577.860,Z 252.125,A 0.000,B 0.000,C 90.000,E1 238.456} C_DIS
LIN {X -0.090,Y -572.561,Z 252.116,A 0.000,B 0.000,C 90.000,E1 236.834} C_DIS
LIN {X 0.182,Y -566.442,Z 252.105,A 0.000,B 0.000,C 90.000,E1 234.895} C_DIS
LIN {X -0.037,Y -562.201,Z 252.097,A 0.000,B 0.000,C 90.000,E1 233.543} C_DIS
LIN {X -0.240,Y -557.041,Z 252.088,A 0.000,B 0.000,C 90.000,E1 231.904} C_DIS
LIN {X 0.066,Y -552.742,Z 252.081,A 0.000,B 0.000,C 90.000,E1 230.481} C_DIS
LIN {X -0.111,Y -549.300,Z 252.074,A 0.000,B 0.000,C 90.000,E1 229.380} C_DIS
LIN {X 0.046,Y -544.874,Z 252.067,A 0.000,B 0.000,C 90.000,E1 227.957} C_DIS
LIN {X 0.079,Y -540.350,Z 252.059,A 0.000,B 0.000,C 90.000,E1 226.539} C_DIS
LIN {X 0.030,Y -535.832,Z 252.051,A 0.000,B 0.000,C 90.000,E1 225.121} C_DIS
LIN {X 0.310,Y -532.175,Z 252.044,A 0.000,B 0.000,C 90.000,E1 223.947} C_DIS
LIN {X 0.011,Y -525.890,Z 252.033,A 0.000,B 0.000,C 90.000,E1 221.962} C_DIS
LIN {X -0.070,Y -518.871,Z 252.020,A 0.000,B 0.000,C 90.000,E1 219.644} C_DIS
LIN {X 0.046,Y -511.958,Z 252.007,A 0.000,B 0.000,C 90.000,E1 217.282} C_DIS
LIN {X -0.060,Y -506.914,Z 251.997,A 0.000,B 0.000,C 90.000,E1 215.518} C_DIS
LIN {X 0.020,Y -501.003,Z 251.986,A 0.000,B 0.000,C 90.000,E1 213.420} C_DIS
LIN {X 0.094,Y -494.523,Z 251.972,A 0.000,B 0.000,C 90.000,E1 211.003} C_DIS
LIN {X 0.073,Y -490.628,Z 251.964,A 0.000,B 0.000,C 90.000,E1 209.489} C_DIS
LIN {X 0.018,Y -484.840,Z 251.950,A 0.000,B 0.000,C 90.000,E1 207.052} C_DIS
LIN {X 0.168,Y -478.293,Z 251.933,A 0.000,B 0.000,C 90.000,E1 203.951} C_DIS
LIN {X -0.041,Y -472.457,Z 251.916,A 0.000,B 0.000,C 90.000,E1 200.865} C_DIS
LIN {X 0.248,Y -467.372,Z 251.899,A 0.000,B 0.000,C 90.000,E1 197.692} C_DIS
LIN {X 0.258,Y -464.159,Z 251.886,A 0.000,B 0.000,C 90.000,E1 195.481} C_DIS
LIN {X -0.086,Y -462.060,Z 251.877,A 0.000,B 0.000,C 90.000,E1 193.939} C_DIS
LIN {X -0.103,Y -459.325,Z 251.865,A 0.000,B 0.000,C 90.000,E1 191.715} C_DIS
LIN {X -0.047,Y -456.359,Z 251.851,A 0.000,B 0.000,C 90.000,E1 189.151} C_DIS
LIN {X -0.218,Y -453.802,Z 251.837,A 0.000,B 0.000,C 90.000,E1 186.606} C_DIS
LIN {X 0.178,Y -451.836,Z 251.824,A 0.000,B 0.000,C 90.000,E1 184.302} C_DIS
LIN {X 0.000,Y -450.086,Z 251.812,A 0.000,B 0.000,C 90.000,E1 182.064} C_DIS
LIN {X 0.208,Y -448.568,Z 251.799,A 0.000,B 0.000,C 90.000,E1 179.771} C_DIS
LIN {X -0.232,Y -447.159,Z 251.783,A 0.000,B 0.000,C 90.000,E1 176.906} C_DIS
LIN {X -0.028,Y -446.425,Z 251.765,A 0.000,B 0.000,C 90.000,E1 173.628} C_DIS
LIN {X -0.047,Y -446.393,Z 251.750,A 0.000,B 0.000,C 90.000,E1 171.027} C_DIS
LIN {X 0.154,Y -446.683,Z 251.739,A 0.000,B 0.000,C 90.000,E1 169.050} C_DIS
LIN {X -0.227,Y -447.652,Z 251.723,A 0.000,B 0.000,C 90.000,E1 166.172} C_DIS
LIN {X 0.039,Y -448.596,Z 251.710,A 0.000,B 0.000,C 90.000,E1 163.866} C_DIS
LIN {X -0.154,Y -449.679,Z 251.700,A 0.000,B 0.000,C 90.000,E1 161.945} C_DIS
LIN {X -0.218,Y -452.163,Z 251.682,A 0.000,B 0.000,C 90.000,E1 158.720} C_DIS
LIN {X 0.105,Y -454.607,Z 251.667,A 0.000,B 0.000,C 90.000,E1 156.102} C_DIS
LIN {X -0.123,Y -457.619,Z 251.653,A 0.000,B 0.000,C 90.000,E1 153.563} C_DIS
LIN {X -0.085,Y -460.169,Z 251.642,A 0.000,B 0.000,C 90.000,E1 151.641} C_DIS
LIN {X 0.186,Y -462.050,Z 251.635,A 0.000,B 0.000,C 90.000,E1 150.333} C_DIS
LIN {X -0.176,Y -464.448,Z 251.627,A 0.000,B 0.000,C 90.000,E1 148.791} C_DIS
LIN {X 0.301,Y -467.469,Z 251.616,A 0.000,B 0.000,C 90.000,E1 146.834} C_DIS
LIN {X 0.061,Y -470.657,Z 251.606,A 0.000,B 0.000,C 90.000,E1 144.975} C_DIS
LIN {X 0.209,Y -472.626,Z 251.599,A 0.000,B 0.000,C 90.000,E1 143.703} C_DIS
LIN {X 0.251,Y -475.520,Z 251.588,A 0.000,B 0.000,C 90.000,E1 141.823} C_DIS
LIN {X -0.017,Y -478.084,Z 251.578,A 0.000,B 0.000,C 90.000,E1 139.989} C_DIS
LIN {X -0.091,Y -479.952,Z 251.569,A 0.000,B 0.000,C 90.000,E1 138.447} C_DIS
LIN {X -0.050,Y -480.897,Z 251.564,A 0.000,B 0.000,C 90.000,E1 137.514} C_DIS
LIN {X -0.201,Y -481.794,Z 251.557,A 0.000,B 0.000,C 90.000,E1 136.296} C_DIS
LIN {X 0.190,Y -482.290,Z 251.552,A 0.000,B 0.000,C 90.000,E1 135.324} C_DIS
LIN {X -0.093,Y -482.616,Z 251.547,A 0.000,B 0.000,C 90.000,E1 134.433} C_DIS
LIN {X -0.025,Y -482.780,Z 251.542,A 0.000,B 0.000,C 90.000,E1 133.500} C_DIS
LIN {X -0.174,Y -482.671,Z 251.535,A 0.000,B 0.000,C 90.000,E1 132.285} C_DIS
LIN {X 0.063,Y -481.975,Z 251.528,A 0.000,B 0.000,C 90.000,E1 131.024} C_DIS
LIN {X 0.048,Y -480.742,Z 251.519,A 0.000,B 0.000,C 90.000,E1 129.483} C_DIS
LIN {X 0.063,Y -479.225,Z 251.511,A 0.000,B 0.000,C 90.000,E1 127.935} C_DIS
LIN {X -0.051,Y -477.753,Z 251.504,A 0.000,B 0.000,C 90.000,E1 126.710} C_DIS
LIN {X 0.196,Y -475.992,Z 251.497,A 0.000,B 0.000,C 90.000,E1 125.438} C_DIS
LIN {X -0.069,Y -473.573,Z 251.488,A 0.000,B 0.000,C 90.000,E1 123.913} C_DIS
LIN {X 0.068,Y -471.990,Z 251.483,A 0.000,B 0.000,C 90.000,E1 122.959} C_DIS
LIN {X -0.045,Y -469.867,Z 251.476,A 0.000,B 0.000,C 90.000,E1 121.720} C_DIS
LIN {X 0.272,Y -466.548,Z 251.466,A 0.000,B 0.000,C 90.000,E1 119.795} C_DIS
LIN {X 0.143,Y -463.767,Z 251.457,A 0.000,B 0.000,C 90.000,E1 118.231} C_DIS
LIN {X -0.008,Y -459.742,Z 251.445,A 0.000,B 0.000,C 90.000,E1 116.027} C_DIS
LIN {X -0.257,Y -456.884,Z 251.436,A 0.000,B 0.000,C 90.000,E1 114.463} C_DIS
LIN {X -0.161,Y -453.002,Z 251.423,A 0.000,B 0.000,C 90.000,E1 112.206} C_DIS
LIN {X -0.150,Y -452.170,Z 251.421,A 0.000,B 0.000,C 90.000,E1 111.716} C_DIS
LIN {X -0.189,Y -452.175,Z 251.421,A 0.000,B 0.000,C 90.000,E1 111.716} C_DIS
LIN {X -0.055,Y -456.917,Z 251.411,A 0.000,B 0.000,C 90.000,E1 109.939} C_DIS
LIN {X -0.154,Y -457.626,Z 251.409,A 0.000,B 0.000,C 90.000,E1 109.631} C_DIS
LIN {X -0.068,Y -466.347,Z 251.386,A 0.000,B 0.000,C 90.000,E1 105.481} C_DIS
LIN {X 0.106,Y -467.879,Z 251.383,A 0.000,B 0.000,C 90.000,E1 104.828} C_DIS
LIN {X 0.134,Y -475.442,Z 251.358,A 0.000,B 0.000,C 90.000,E1 100.433} C_DIS
LIN {X -0.028,Y -476.092,Z 251.356,A 0.000,B 0.000,C 90.000,E1 100.141} C_DIS
LIN {X -0.224,Y -482.012,Z 251.331,A 0.000,B 0.000,C 90.000,E1 95.511} C_DIS
LIN {X 0.047,Y -482.683,Z 251.324,A 0.000,B 0.000,C 90.000,E1 94.245} C_DIS
LIN {X 0.047,Y -485.455,Z 251.305,A 0.000,B 0.000,C 90.000,E1 90.859} C_DIS
LIN {X 0.010,Y -485.500,Z 251.300,A 0.000,B 0.000,C 90.000,E1 89.943} C_DIS
LIN {X 0.079,Y -486.383,Z 251.281,A 0.000,B 0.000,C 90.000,E1 86.560} C_DIS
LIN {X -0.096,Y -486.365,Z 251.279,A 0.000,B 0.000,C 90.000,E1 86.274} C_DIS
LIN {X -0.008,Y -484.690,Z 251.254,A 0.000,B 0.000,C 90.000,E1 81.659} C_DIS
LIN {X 0.138,Y -484.067,Z 251.250,A 0.000,B 0.000,C 90.000,E1 81.027} C_DIS
LIN {X -0.206,Y -480.637,Z 251.228,A 0.000,B 0.000,C 90.000,E1 77.061} C_DIS
LIN {X 0.228,Y -480.337,Z 251.226,A 0.000,B 0.000,C 90.000,E1 76.700} C_DIS
LIN {X 0.131,Y -474.147,Z 251.200,A 0.000,B 0.000,C 90.000,E1 72.054} C_DIS
LIN {X -0.017,Y -466.402,Z 251.176,A 0.000,B 0.000,C 90.000,E1 67.614} C_DIS
LIN {X -0.058,Y -466.400,Z 251.176,A 0.000,B 0.000,C 90.000,E1 67.614} C_DIS
LIN {X -0.071,Y -471.878,Z 251.164,A 0.000,B 0.000,C 90.000,E1 65.485} C_DIS
LIN {X 0.137,Y -475.935,Z 251.155,A 0.000,B 0.000,C 90.000,E1 63.896} C_DIS
LIN {X -0.251,Y -481.668,Z 251.143,A 0.000,B 0.000,C 90.000,E1 61.769} C_DIS
LIN {X -0.023,Y -487.564,Z 251.131,A 0.000,B 0.000,C 90.000,E1 59.587} C_DIS
LIN {X 0.027,Y -490.174,Z 251.126,A 0.000,B 0.000,C 90.000,E1 58.663} C_DIS
LIN {X 0.202,Y -494.426,Z 251.118,A 0.000,B 0.000,C 90.000,E1 57.120} C_DIS
LIN {X 0.035,Y -497.690,Z 251.111,A 0.000,B 0.000,C 90.000,E1 55.928} C_DIS
LIN {X 0.208,Y -501.517,Z 251.102,A 0.000,B 0.000,C 90.000,E1 54.402} C_DIS
LIN {X 0.147,Y -504.427,Z 251.096,A 0.000,B 0.000,C 90.000,E1 53.210} C_DIS
LIN {X 0.029,Y -507.106,Z 251.089,A 0.000,B 0.000,C 90.000,E1 52.029} C_DIS
LIN {X -0.268,Y -508.928,Z 251.084,A 0.000,B 0.000,C 90.000,E1 51.170} C_DIS
LIN {X -0.320,Y -511.130,Z 251.078,A 0.000,B 0.000,C 90.000,E1 49.989} C_DIS
LIN {X 0.078,Y -512.607,Z 251.073,A 0.000,B 0.000,C 90.000,E1 49.057} C_DIS
LIN {X 0.159,Y -513.929,Z 251.068,A 0.000,B 0.000,C 90.000,E1 48.162} C_DIS
LIN {X -0.132,Y -515.033,Z 251.063,A 0.000,B 0.000,C 90.000,E1 47.310} C_DIS
LIN {X -0.144,Y -516.256,Z 251.056,A 0.000,B 0.000,C 90.000,E1 46.134} C_DIS
LIN {X 0.221,Y -517.048,Z 251.050,A 0.000,B 0.000,C 90.000,E1 44.919} C_DIS
LIN {X 0.320,Y -517.532,Z 251.045,A 0.000,B 0.000,C 90.000,E1 44.028} C_DIS
LIN {X -0.035,Y -517.905,Z 251.038,A 0.000,B 0.000,C 90.000,E1 42.894} C_DIS
LIN {X 0.096,Y -518.041,Z 251.033,A 0.000,B 0.000,C 90.000,E1 42.000} C_DIS
LIN {X -0.152,Y -518.000,Z 251.029,A 0.000,B 0.000,C 90.000,E1 41.148} C_DIS
LIN {X 0.259,Y -517.655,Z 251.022,A 0.000,B 0.000,C 90.000,E1 39.930} C_DIS
LIN {X 0.008,Y -517.018,Z 251.016,A 0.000,B 0.000,C 90.000,E1 38.785} C_DIS
LIN {X 0.139,Y -516.421,Z 251.011,A 0.000,B 0.000,C 90.000,E1 37.890} C_DIS
LIN {X -0.055,Y -515.594,Z 251.006,A 0.000,B 0.000,C 90.000,E1 37.030} C_DIS
LIN {X 0.047,Y -514.582,Z 251.001,A 0.000,B 0.000,C 90.000,E1 36.137} C_DIS
LIN {X 0.168,Y -512.998,Z 250.994,A 0.000,B 0.000,C 90.000,E1 34.945} C_DIS
LIN {X -0.108,Y -510.819,Z 250.986,A 0.000,B 0.000,C 90.000,E1 33.499} C_DIS
LIN {X -0.094,Y -508.188,Z 250.976,A 0.000,B 0.000,C 90.000,E1 31.720} C_DIS
LIN {X 0.032,Y -504.402,Z 250.961,A 0.000,B 0.000,C 90.000,E1 29.027} C_DIS
LIN {X 0.185,Y -501.389,Z 250.948,A 0.000,B 0.000,C 90.000,E1 26.616} C_DIS
LIN {X 0.177,Y -499.074,Z 250.936,A 0.000,B 0.000,C 90.000,E1 24.515} C_DIS
LIN {X -0.300,Y -496.939,Z 250.925,A 0.000,B 0.000,C 90.000,E1 22.461} C_DIS
LIN {X 0.089,Y -494.991,Z 250.913,A 0.000,B 0.000,C 90.000,E1 20.301} C_DIS
LIN {X 0.082,Y -493.178,Z 250.901,A 0.000,B 0.000,C 90.000,E1 18.181} C_DIS
LIN {X -0.152,Y -491.719,Z 250.891,A 0.000,B 0.000,C 90.000,E1 16.386} C_DIS
LIN {X -0.049,Y -490.018,Z 250.877,A 0.000,B 0.000,C 90.000,E1 13.939} C_DIS
LIN {X 0.003,Y -488.446,Z 250.862,A 0.000,B 0.000,C 90.000,E1 11.186} C_DIS
LIN {X 0.149,Y -487.664,Z 250.850,A 0.000,B 0.000,C 90.000,E1 9.029} C_DIS
LIN {X -0.066,Y -487.047,Z 250.837,A 0.000,B 0.000,C 90.000,E1 6.606} C_DIS
LIN {X -0.161,Y -486.873,Z 250.825,A 0.000,B 0.000,C 90.000,E1 4.473} C_DIS
LIN {X -0.174,Y -487.166,Z 250.809,A 0.000,B 0.000,C 90.000,E1 1.718} C_DIS
LIN {X -0.193,Y -487.343,Z 250.804,A 0.000,B 0.000,C 90.000,E1 0.802} C_DIS
LIN {X 0.182,Y -488.701,Z 250.789,A 0.000,B 0.000,C 90.000,E1 357.936} C_DIS
LIN {X -0.096,Y -490.502,Z 250.775,A 0.000,B 0.000,C 90.000,E1 355.527} C_DIS
LIN {X -0.221,Y -495.904,Z 250.748,A 0.000,B 0.000,C 90.000,E1 350.679} C_DIS
LIN {X 0.241,Y -499.307,Z 250.738,A 0.000,B 0.000,C 90.000,E1 348.814} C_DIS
LIN {X 0.130,Y -509.438,Z 250.716,A 0.000,B 0.000,C 90.000,E1 344.936} C_DIS
LIN {X 0.181,Y -513.466,Z 250.708,A 0.000,B 0.000,C 90.000,E1 343.449} C_DIS
LIN {X 0.064,Y -519.168,Z 250.697,A 0.000,B 0.000,C 90.000,E1 341.402} C_DIS
LIN {X 0.283,Y -528.274,Z 250.681,A 0.000,B 0.000,C 90.000,E1 338.465} C_DIS
LIN {X 0.222,Y -534.154,Z 250.671,A 0.000,B 0.000,C 90.000,E1 336.741} C_DIS
LIN {X -0.003,Y -540.144,Z 250.661,A 0.000,B 0.000,C 90.000,E1 335.049} C_DIS
LIN {X -0.123,Y -548.333,Z 250.649,A 0.000,B 0.000,C 90.000,E1 332.794} C_DIS
LIN {X -0.077,Y -553.639,Z 250.641,A 0.000,B 0.000,C 90.000,E1 331.385} C_DIS
LIN {X -0.164,Y -558.862,Z 250.633,A 0.000,B 0.000,C 90.000,E1 329.999} C_DIS
LIN {X -0.162,Y -563.847,Z 250.626,A 0.000,B 0.000,C 90.000,E1 328.614} C_DIS
LIN {X -0.336,Y -570.785,Z 250.615,A 0.000,B 0.000,C 90.000,E1 326.707} C_DIS
LIN {X -0.168,Y -577.053,Z 250.606,A 0.000,B 0.000,C 90.000,E1 325.055} C_DIS
LIN {X -0.347,Y -581.173,Z 250.600,A 0.000,B 0.000,C 90.000,E1 323.989} C_DIS
LIN {X 0.351,Y -584.987,Z 250.594,A 0.000,B 0.000,C 90.000,E1 322.844} C_DIS
LIN {X -0.180,Y -588.567,Z 250.588,A 0.000,B 0.000,C 90.000,E1 321.823} C_DIS
LIN {X 0.343,Y -594.865,Z 250.577,A 0.000,B 0.000,C 90.000,E1 319.908} C_DIS
LIN {X 0.113,Y -601.548,Z 250.567,A 0.000,B 0.000,C 90.000,E1 318.081} C_DIS
LIN {X -0.025,Y -606.309,Z 250.560,A 0.000,B 0.000,C 90.000,E1 316.782} C_DIS
LIN {X 0.072,Y -610.025,Z 250.554,A 0.000,B 0.000,C 90.000,E1 315.729} C_DIS
LIN {X -0.034,Y -612.581,Z 250.550,A 0.000,B 0.000,C 90.000,E1 314.960} C_DIS
LIN {X -0.114,Y -614.887,Z 250.545,A 0.000,B 0.000,C 90.000,E1 314.190} C_DIS
LIN {X 0.100,Y -617.587,Z 250.540,A 0.000,B 0.000,C 90.000,E1 313.137} C_DIS
LIN {X 0.078,Y -619.426,Z 250.535,A 0.000,B 0.000,C 90.000,E1 312.366} C_DIS
LIN {X 0.077,Y -621.032,Z 250.531,A 0.000,B 0.000,C 90.000,E1 311.595} C_DIS
LIN {X 0.090,Y -622.516,Z 250.527,A 0.000,B 0.000,C 90.000,E1 310.825} C_DIS
LIN {X 0.044,Y -624.291,Z 250.521,A 0.000,B 0.000,C 90.000,E1 309.806} C_DIS
LIN {X 0.084,Y -625.516,Z 250.517,A 0.000,B 0.000,C 90.000,E1 309.036} C_DIS
LIN {X 0.083,Y -626.854,Z 250.511,A 0.000,B 0.000,C 90.000,E1 308.016} C_DIS
LIN {X 0.248,Y -627.735,Z 250.507,A 0.000,B 0.000,C 90.000,E1 307.237} C_DIS
LIN {X 0.073,Y -628.266,Z 250.504,A 0.000,B 0.000,C 90.000,E1 306.744} C_DIS
LIN {X 0.104,Y -628.853,Z 250.499,A 0.000,B 0.000,C 90.000,E1 305.724} C_DIS
LIN {X -0.232,Y -629.180,Z 250.493,A 0.000,B 0.000,C 90.000,E1 304.739} C_DIS
LIN {X -0.398,Y -629.316,Z 250.489,A 0.000,B 0.000,C 90.000,E1 303.992} C_DIS
LIN {X -0.208,Y -629.168,Z 250.483,A 0.000,B 0.000,C 90.000,E1 302.959} C_DIS
LIN {X -0.369,Y -628.688,Z 250.479,A 0.000,B 0.000,C 90.000,E1 302.212} C_DIS
LIN {X 0.000,Y -627.843,Z 250.475,A 0.000,B 0.000,C 90.000,E1 301.416} C_DIS
LIN {X 0.154,Y -626.448,Z 250.469,A 0.000,B 0.000,C 90.000,E1 300.384} C_DIS
LIN {X 0.175,Y -625.531,Z 250.466,A 0.000,B 0.000,C 90.000,E1 299.873} C_DIS
LIN {X -0.029,Y -623.549,Z 250.460,A 0.000,B 0.000,C 90.000,E1 298.871} C_DIS
LIN {X -0.016,Y -621.816,Z 250.456,A 0.000,B 0.000,C 90.000,E1 298.103} C_DIS
LIN {X -0.017,Y -619.272,Z 250.450,A 0.000,B 0.000,C 90.000,E1 297.078} C_DIS
LIN {X -0.063,Y -615.935,Z 250.443,A 0.000,B 0.000,C 90.000,E1 295.796} C_DIS
LIN {X -0.003,Y -609.694,Z 250.430,A 0.000,B 0.000,C 90.000,E1 293.462} C_DIS
LIN {X 0.174,Y -603.895,Z 250.417,A 0.000,B 0.000,C 90.000,E1 291.099} C_DIS
LIN {X -0.173,Y -599.041,Z 250.406,A 0.000,B 0.000,C 90.000,E1 289.033} C_DIS
LIN {X 0.317,Y -592.855,Z 250.390,A 0.000,B 0.000,C 90.000,E1 286.079} C_DIS
LIN {X -0.269,Y -588.911,Z 250.378,A 0.000,B 0.000,C 90.000,E1 284.008} C_DIS
LIN {X 0.102,Y -584.813,Z 250.363,A 0.000,B 0.000,C 90.000,E1 281.299} C_DIS
LIN {X 0.124,Y -581.350,Z 250.346,A 0.000,B 0.000,C 90.000,E1 278.341} C_DIS
LIN {X 0.162,Y -579.311,Z 250.333,A 0.000,B 0.000,C 90.000,E1 275.910} C_DIS
LIN {X -0.121,Y -577.700,Z 250.315,A 0.000,B 0.000,C 90.000,E1 272.694} C_DIS
LIN {X -0.043,Y -577.935,Z 250.292,A 0.000,B 0.000,C 90.000,E1 268.625} C_DIS
LIN {X 0.152,Y -580.664,Z 250.270,A 0.000,B 0.000,C 90.000,E1 264.552} C_DIS
LIN {X 0.134,Y -583.355,Z 250.256,A 0.000,B 0.000,C 90.000,E1 262.129} C_DIS
LIN {X -0.200,Y -586.612,Z 250.243,A 0.000,B 0.000,C 90.000,E1 259.746} C_DIS
LIN {X -0.007,Y -589.916,Z 250.231,A 0.000,B 0.000,C 90.000,E1 257.589} C_DIS
LIN {X -0.009,Y -592.343,Z 250.222,A 0.000,B 0.000,C 90.000,E1 255.992} C_DIS
LIN {X -0.224,Y -594.373,Z 250.215,A 0.000,B 0.000,C 90.000,E1 254.685} C_DIS
LIN {X 0.163,Y -596.040,Z 250.207,A 0.000,B 0.000,C 90.000,E1 253.323} C_DIS
LIN {X 0.016,Y -596.786,Z 250.203,A 0.000,B 0.000,C 90.000,E1 252.543} C_DIS
LIN {X -0.125,Y -597.292,Z 250.199,A 0.000,B 0.000,C 90.000,E1 251.764} C_DIS
LIN {X 0.194,Y -597.613,Z 250.193,A 0.000,B 0.000,C 90.000,E1 250.678} C_DIS
LIN {X -0.048,Y -597.751,Z 250.187,A 0.000,B 0.000,C 90.000,E1 249.645} C_DIS
LIN {X 0.014,Y -597.604,Z 250.183,A 0.000,B 0.000,C 90.000,E1 248.847} C_DIS
LIN {X 0.074,Y -597.176,Z 250.178,A 0.000,B 0.000,C 90.000,E1 248.050} C_DIS
LIN {X -0.194,Y -596.454,Z 250.174,A 0.000,B 0.000,C 90.000,E1 247.283} C_DIS
LIN {X -0.233,Y -595.170,Z 250.168,A 0.000,B 0.000,C 90.000,E1 246.230} C_DIS
LIN {X 0.039,Y -593.929,Z 250.163,A 0.000,B 0.000,C 90.000,E1 245.409} C_DIS
LIN {X 0.298,Y -592.435,Z 250.159,A 0.000,B 0.000,C 90.000,E1 244.588} C_DIS
LIN {X -0.092,Y -590.194,Z 250.153,A 0.000,B 0.000,C 90.000,E1 243.563} C_DIS
LIN {X 0.012,Y -587.582,Z 250.147,A 0.000,B 0.000,C 90.000,E1 242.487} C_DIS
LIN {X -0.172,Y -584.886,Z 250.141,A 0.000,B 0.000,C 90.000,E1 241.435} C_DIS
LIN {X 0.251,Y -582.743,Z 250.137,A 0.000,B 0.000,C 90.000,E1 240.589} C_DIS
LIN {X -0.141,Y -578.855,Z 250.129,A 0.000,B 0.000,C 90.000,E1 239.282} C_DIS
LIN {X -0.151,Y -575.415,Z 250.123,A 0.000,B 0.000,C 90.000,E1 238.201} C_DIS
LIN {X 0.060,Y -570.092,Z 250.114,A 0.000,B 0.000,C 90.000,E1 236.548} C_DIS
LIN {X 0.161,Y -564.875,Z 250.105,A 0.000,B 0.000,C 90.000,E1 234.895} C_DIS
LIN {X -0.086,Y -560.612,Z 250.097,A 0.000,B 0.000,C 90.000,E1 233.543} C_DIS
LIN {X 0.037,Y -556.316,Z 250.090,A 0.000,B 0.000,C 90.000,E1 232.145} C_DIS
LIN {X 0.319,Y -551.992,Z 250.082,A 0.000,B 0.000,C 90.000,E1 230.723} C_DIS
LIN {X -0.243,Y -547.645,Z 250.074,A 0.000,B 0.000,C 90.000,E1 229.380} C_DIS
LIN {X -0.130,Y -542.274,Z 250.065,A 0.000,B 0.000,C 90.000,E1 227.676} C_DIS
LIN {X -0.133,Y -536.856,Z 250.055,A 0.000,B 0.000,C 90.000,E1 225.972} C_DIS
LIN {X 0.136,Y -532.330,Z 250.047,A 0.000,B 0.000,C 90.000,E1 224.514} C_DIS
LIN {X 0.162,Y -525.034,Z 250.035,A 0.000,B 0.000,C 90.000,E1 222.204} C_DIS
LIN {X 0.172,Y -519.719,Z 250.025,A 0.000,B 0.000,C 90.000,E1 220.458} C_DIS
LIN {X 0.331,Y -517.145,Z 250.020,A 0.000,B 0.000,C 90.000,E1 219.564} C_DIS
LIN {X 0.079,Y -510.235,Z 250.007,A 0.000,B 0.000,C 90.000,E1 217.237} C_DIS
LIN {X -0.273,Y -506.897,Z 250.000,A 0.000,B 0.000,C 90.000,E1 216.091} C_DIS
LIN {X -0.184,Y -500.951,Z 249.989,A 0.000,B 0.000,C 90.000,E1 213.992} C_DIS
LIN {X -0.113,Y -495.179,Z 249.977,A 0.000,B 0.000,C 90.000,E1 211.878} C_DIS
LIN {X -0.039,Y -490.468,Z 249.967,A 0.000,B 0.000,C 90.000,E1 210.050} C_DIS
LIN {X -0.118,Y -483.116,Z 249.950,A 0.000,B 0.000,C 90.000,E1 207.001} C_DIS
LIN {X -0.002,Y -477.196,Z 249.935,A 0.000,B 0.000,C 90.000,E1 204.207} C_DIS
LIN {X 0.026,Y -472.973,Z 249.922,A 0.000,B 0.000,C 90.000,E1 202.025} C_DIS
LIN {X 0.246,Y -469.717,Z 249.912,A 0.000,B 0.000,C 90.000,E1 200.120} C_DIS
LIN {X -0.043,Y -465.749,Z 249.898,A 0.000,B 0.000,C 90.000,E1 197.638} C_DIS
LIN {X -0.068,Y -462.581,Z 249.886,A 0.000,B 0.000,C 90.000,E1 195.426} C_DIS
LIN {X 0.011,Y -460.470,Z 249.877,A 0.000,B 0.000,C 90.000,E1 193.828} C_DIS
LIN {X 0.050,Y -457.734,Z 249.864,A 0.000,B 0.000,C 90.000,E1 191.591} C_DIS
LIN {X -0.173,Y -455.156,Z 249.852,A 0.000,B 0.000,C 90.000,E1 189.378} C_DIS
LIN {X -0.150,Y -452.865,Z 249.840,A 0.000,B 0.000,C 90.000,E1 187.125} C_DIS
LIN {X -0.230,Y -450.825,Z 249.827,A 0.000,B 0.000,C 90.000,E1 184.878} C_DIS
LIN {X 0.160,Y -449.519,Z 249.818,A 0.000,B 0.000,C 90.000,E1 183.212} C_DIS
LIN {X -0.082,Y -447.860,Z 249.805,A 0.000,B 0.000,C 90.000,E1 180.974} C_DIS
LIN {X 0.198,Y -446.344,Z 249.791,A 0.000,B 0.000,C 90.000,E1 178.339} C_DIS
LIN {X 0.035,Y -445.356,Z 249.776,A 0.000,B 0.000,C 90.000,E1 175.755} C_DIS
LIN {X -0.114,Y -444.957,Z 249.762,A 0.000,B 0.000,C 90.000,E1 173.166} C_DIS
LIN {X 0.244,Y -445.158,Z 249.744,A 0.000,B 0.000,C 90.000,E1 169.859} C_DIS
LIN {X 0.069,Y -446.229,Z 249.724,A 0.000,B 0.000,C 90.000,E1 166.297} C_DIS
LIN {X 0.145,Y -447.358,Z 249.710,A 0.000,B 0.000,C 90.000,E1 163.685} C_DIS
LIN {X -0.075,Y -448.434,Z 249.699,A 0.000,B 0.000,C 90.000,E1 161.764} C_DIS
LIN {X -0.188,Y -450.977,Z 249.681,A 0.000,B 0.000,C 90.000,E1 158.539} C_DIS
LIN {X 0.094,Y -453.434,Z 249.666,A 0.000,B 0.000,C 90.000,E1 155.921} C_DIS
LIN {X -0.178,Y -456.514,Z 249.652,A 0.000,B 0.000,C 90.000,E1 153.384} C_DIS
LIN {X 0.179,Y -460.527,Z 249.636,A 0.000,B 0.000,C 90.000,E1 150.461} C_DIS
LIN {X 0.187,Y -462.920,Z 249.627,A 0.000,B 0.000,C 90.000,E1 148.869} C_DIS
LIN {X -0.021,Y -465.926,Z 249.617,A 0.000,B 0.000,C 90.000,E1 146.993} C_DIS
LIN {X -0.037,Y -469.125,Z 249.606,A 0.000,B 0.000,C 90.000,E1 145.102} C_DIS
LIN {X -0.135,Y -471.579,Z 249.597,A 0.000,B 0.000,C 90.000,E1 143.543} C_DIS
LIN {X -0.191,Y -473.977,Z 249.589,A 0.000,B 0.000,C 90.000,E1 141.984} C_DIS
LIN {X -0.290,Y -476.142,Z 249.580,A 0.000,B 0.000,C 90.000,E1 140.436} C_DIS
LIN {X -0.147,Y -477.699,Z 249.573,A 0.000,B 0.000,C 90.000,E1 139.175} C_DIS
LIN {X -0.026,Y -479.068,Z 249.566,A 0.000,B 0.000,C 90.000,E1 137.919} C_DIS
LIN {X -0.116,Y -479.637,Z 249.563,A 0.000,B 0.000,C 90.000,E1 137.310} C_DIS
LIN {X 0.040,Y -480.487,Z 249.556,A 0.000,B 0.000,C 90.000,E1 136.053} C_DIS
LIN {X -0.263,Y -480.951,Z 249.551,A 0.000,B 0.000,C 90.000,E1 135.162} C_DIS
LIN {X 0.119,Y -481.264,Z 249.546,A 0.000,B 0.000,C 90.000,E1 134.190} C_DIS
LIN {X -0.178,Y -481.400,Z 249.540,A 0.000,B 0.000,C 90.000,E1 133.299} C_DIS
LIN {X -0.002,Y -481.170,Z 249.534,A 0.000,B 0.000,C 90.000,E1 132.043} C_DIS
LIN {X -0.272,Y -480.638,Z 249.528,A 0.000,B 0.000,C 90.000,E1 131.148} C_DIS
LIN {X 0.051,Y -479.426,Z 249.520,A 0.000,B 0.000,C 90.000,E1 129.564} C_DIS
LIN {X -0.056,Y -478.267,Z 249.513,A 0.000,B 0.000,C 90.000,E1 128.338} C_DIS
LIN {X 0.024,Y -477.270,Z 249.508,A 0.000,B 0.000,C 90.000,E1 127.397} C_DIS
LIN {X 0.093,Y -476.103,Z 249.503,A 0.000,B 0.000,C 90.000,E1 126.457} C_DIS
LIN {X -0.066,Y -474.349,Z 249.496,A 0.000,B 0.000,C 90.000,E1 125.231} C_DIS
LIN {X 0.034,Y -471.930,Z 249.487,A 0.000,B 0.000,C 90.000,E1 123.658} C_DIS
LIN {X -0.142,Y -468.730,Z 249.477,A 0.000,B 0.000,C 90.000,E1 121.799} C_DIS
LIN {X 0.154,Y -465.419,Z 249.466,A 0.000,B 0.000,C 90.000,E1 119.873} C_DIS
LIN {X 0.011,Y -462.631,Z 249.457,A 0.000,B 0.000,C 90.000,E1 118.309} C_DIS
LIN {X -0.161,Y -458.602,Z 249.445,A 0.000,B 0.000,C 90.000,E1 116.104} C_DIS
LIN {X 0.178,Y -455.747,Z 249.436,A 0.000,B 0.000,C 90.000,E1 114.463} C_DIS
LIN {X 0.241,Y -451.865,Z 249.424,A 0.000,B 0.000,C 90.000,E1 112.206} C_DIS
LIN {X 0.138,Y -451.449,Z 249.422,A 0.000,B 0.000,C 90.000,E1 111.972} C_DIS
LIN {X 0.098,Y -451.440,Z 249.422,A 0.000,B 0.000,C 90.000,E1 111.972} C_DIS
LIN {X -0.095,Y -456.777,Z 249.411,A 0.000,B 0.000,C 90.000,E1 109.993} C_DIS
LIN {X 0.236,Y -457.538,Z 249.409,A 0.000,B 0.000,C 90.000,E1 109.631} C_DIS
LIN {X -0.125,Y -466.229,Z 249.386,A 0.000,B 0.000,C 90.000,E1 105.536} C_DIS
LIN {X -0.073,Y -467.790,Z 249.383,A 0.000,B 0.000,C 90.000,E1 104.898} C_DIS
LIN {X -0.102,Y -475.996,Z 249.357,A 0.000,B 0.000,C 90.000,E1 100.197} C_DIS
LIN {X 0.047,Y -476.691,Z 249.353,A 0.000,B 0.000,C 90.000,E1 99.557} C_DIS
LIN {X 0.171,Y -481.936,Z 249.331,A 0.000,B 0.000,C 90.000,E1 95.511} C_DIS
LIN {X 0.020,Y -482.208,Z 249.329,A 0.000,B 0.000,C 90.000,E1 95.220} C_DIS
LIN {X -0.042,Y -485.404,Z 249.305,A 0.000,B 0.000,C 90.000,E1 90.917} C_DIS
LIN {X -0.217,Y -485.528,Z 249.303,A 0.000,B 0.000,C 90.000,E1 90.630} C_DIS
LIN {X -0.010,Y -486.365,Z 249.281,A 0.000,B 0.000,C 90.000,E1 86.617} C_DIS
LIN {X -0.185,Y -486.367,Z 249.280,A 0.000,B 0.000,C 90.000,E1 86.331} C_DIS
LIN {X 0.149,Y -485.675,Z 249.273,A 0.000,B 0.000,C 90.000,E1 85.065} C_DIS
LIN {X -0.161,Y -484.692,Z 249.254,A 0.000,B 0.000,C 90.000,E1 81.724} C_DIS
LIN {X 0.186,Y -484.489,Z 249.252,A 0.000,B 0.000,C 90.000,E1 81.376} C_DIS
LIN {X 0.189,Y -480.663,Z 249.228,A 0.000,B 0.000,C 90.000,E1 77.061} C_DIS
LIN {X 0.155,Y -480.417,Z 249.227,A 0.000,B 0.000,C 90.000,E1 76.756} C_DIS
LIN {X -0.072,Y -474.194,Z 249.201,A 0.000,B 0.000,C 90.000,E1 72.127} C_DIS
LIN {X -0.138,Y -473.020,Z 249.197,A 0.000,B 0.000,C 90.000,E1 71.511} C_DIS
LIN {X -0.085,Y -465.966,Z 249.174,A 0.000,B 0.000,C 90.000,E1 67.305} C_DIS
LIN {X 0.055,Y -465.968,Z 249.174,A 0.000,B 0.000,C 90.000,E1 67.283} C_DIS
LIN {X -0.178,Y -471.310,Z 249.162,A 0.000,B 0.000,C 90.000,E1 65.229} C_DIS
LIN {X 0.019,Y -475.343,Z 249.154,A 0.000,B 0.000,C 90.000,E1 63.640} C_DIS
LIN {X 0.063,Y -480.270,Z 249.143,A 0.000,B 0.000,C 90.000,E1 61.769} C_DIS
LIN {X 0.010,Y -486.157,Z 249.131,A 0.000,B 0.000,C 90.000,E1 59.616} C_DIS
LIN {X -0.139,Y -489.589,Z 249.124,A 0.000,B 0.000,C 90.000,E1 58.408} C_DIS
LIN {X 0.028,Y -492.997,Z 249.118,A 0.000,B 0.000,C 90.000,E1 57.168} C_DIS
LIN {X -0.023,Y -496.270,Z 249.111,A 0.000,B 0.000,C 90.000,E1 55.960} C_DIS
LIN {X -0.295,Y -500.095,Z 249.103,A 0.000,B 0.000,C 90.000,E1 54.482} C_DIS
LIN {X 0.207,Y -503.661,Z 249.094,A 0.000,B 0.000,C 90.000,E1 52.924} C_DIS
LIN {X 0.078,Y -506.319,Z 249.088,A 0.000,B 0.000,C 90.000,E1 51.743} C_DIS
LIN {X -0.007,Y -508.593,Z 249.081,A 0.000,B 0.000,C 90.000,E1 50.561} C_DIS
LIN {X -0.061,Y -510.691,Z 249.074,A 0.000,B 0.000,C 90.000,E1 49.380} C_DIS
LIN {X 0.245,Y -512.458,Z 249.068,A 0.000,B 0.000,C 90.000,E1 48.162} C_DIS
LIN {X -0.062,Y -513.559,Z 249.063,A 0.000,B 0.000,C 90.000,E1 47.310} C_DIS
LIN {X -0.004,Y -514.478,Z 249.058,A 0.000,B 0.000,C 90.000,E1 46.419} C_DIS
LIN {X -0.291,Y -515.218,Z 249.053,A 0.000,B 0.000,C 90.000,E1 45.567} C_DIS
LIN {X 0.058,Y -515.924,Z 249.046,A 0.000,B 0.000,C 90.000,E1 44.352} C_DIS
LIN {X 0.060,Y -516.342,Z 249.040,A 0.000,B 0.000,C 90.000,E1 43.176} C_DIS
LIN {X 0.144,Y -516.543,Z 249.035,A 0.000,B 0.000,C 90.000,E1 42.285} C_DIS
LIN {X -0.195,Y -516.514,Z 249.029,A 0.000,B 0.000,C 90.000,E1 41.148} C_DIS
LIN {X 0.193,Y -516.161,Z 249.022,A 0.000,B 0.000,C 90.000,E1 39.930} C_DIS
LIN {X 0.242,Y -515.499,Z 249.015,A 0.000,B 0.000,C 90.000,E1 38.749} C_DIS
LIN {X 0.035,Y -514.873,Z 249.011,A 0.000,B 0.000,C 90.000,E1 37.890} C_DIS
LIN {X 0.134,Y -514.015,Z 249.006,A 0.000,B 0.000,C 90.000,E1 36.996} C_DIS
LIN {X -0.091,Y -512.974,Z 249.001,A 0.000,B 0.000,C 90.000,E1 36.137} C_DIS
LIN {X 0.006,Y -511.365,Z 248.994,A 0.000,B 0.000,C 90.000,E1 34.945} C_DIS
LIN {X 0.032,Y -508.667,Z 248.984,A 0.000,B 0.000,C 90.000,E1 33.166} C_DIS
LIN {X -0.001,Y -505.976,Z 248.974,A 0.000,B 0.000,C 90.000,E1 31.386} C_DIS
LIN {X -0.009,Y -502.573,Z 248.961,A 0.000,B 0.000,C 90.000,E1 28.999} C_DIS
LIN {X -0.154,Y -499.560,Z 248.948,A 0.000,B 0.000,C 90.000,E1 26.616} C_DIS
LIN {X 0.187,Y -497.591,Z 248.938,A 0.000,B 0.000,C 90.000,E1 24.771} C_DIS
LIN {X -0.133,Y -495.439,Z 248.926,A 0.000,B 0.000,C 90.000,E1 22.695} C_DIS
LIN {X 0.033,Y -493.457,Z 248.914,A 0.000,B 0.000,C 90.000,E1 20.556} C_DIS
LIN {X 0.149,Y -491.639,Z 248.902,A 0.000,B 0.000,C 90.000,E1 18.417} C_DIS
LIN {X -0.122,Y -490.194,Z 248.892,A 0.000,B 0.000,C 90.000,E1 16.622} C_DIS
LIN {X 0.045,Y -488.797,Z 248.882,A 0.000,B 0.000,C 90.000,E1 14.773} C_DIS
LIN {X 0.172,Y -488.028,Z 248.875,A 0.000,B 0.000,C 90.000,E1 13.536} C_DIS
LIN {X -0.188,Y -486.657,Z 248.862,A 0.000,B 0.000,C 90.000,E1 11.130} C_DIS
LIN {X -0.086,Y -485.911,Z 248.850,A 0.000,B 0.000,C 90.000,E1 8.973} C_DIS
LIN {X -0.160,Y -485.309,Z 248.838,A 0.000,B 0.000,C 90.000,E1 6.834} C_DIS
LIN {X 0.176,Y -485.092,Z 248.826,A 0.000,B 0.000,C 90.000,E1 4.645} C_DIS
LIN {X -0.078,Y -485.380,Z 248.809,A 0.000,B 0.000,C 90.000,E1 1.604} C_DIS
LIN {X -0.117,Y -485.539,Z 248.804,A 0.000,B 0.000,C 90.000,E1 0.688} C_DIS
LIN {X -0.191,Y -486.662,Z 248.790,A 0.000,B 0.000,C 90.000,E1 358.282} C_DIS
LIN {X -0.193,Y -488.649,Z 248.775,A 0.000,B 0.000,C 90.000,E1 355.527} C_DIS
LIN {X 0.055,Y -494.003,Z 248.748,A 0.000,B 0.000,C 90.000,E1 350.622} C_DIS
LIN {X -0.016,Y -497.436,Z 248.738,A 0.000,B 0.000,C 90.000,E1 348.814} C_DIS
LIN {X -0.163,Y -506.835,Z 248.718,A 0.000,B 0.000,C 90.000,E1 345.227} C_DIS
LIN {X -0.158,Y -510.909,Z 248.710,A 0.000,B 0.000,C 90.000,E1 343.740} C_DIS
LIN {X 0.155,Y -516.609,Z 248.698,A 0.000,B 0.000,C 90.000,E1 341.638} C_DIS
LIN {X -0.226,Y -526.521,Z 248.680,A 0.000,B 0.000,C 90.000,E1 338.465} C_DIS
LIN {X -0.122,Y -532.439,Z 248.671,A 0.000,B 0.000,C 90.000,E1 336.719} C_DIS
LIN {X 0.115,Y -538.451,Z 248.661,A 0.000,B 0.000,C 90.000,E1 334.973} C_DIS
LIN {X -0.291,Y -546.667,Z 248.648,A 0.000,B 0.000,C 90.000,E1 332.743} C_DIS
LIN {X -0.019,Y -551.979,Z 248.641,A 0.000,B 0.000,C 90.000,E1 331.307} C_DIS
LIN {X -0.129,Y -557.231,Z 248.633,A 0.000,B 0.000,C 90.000,E1 329.921} C_DIS
LIN {X -0.150,Y -562.237,Z 248.625,A 0.000,B 0.000,C 90.000,E1 328.535} C_DIS
LIN {X 0.117,Y -569.212,Z 248.614,A 0.000,B 0.000,C 90.000,E1 326.580} C_DIS
LIN {X -0.221,Y -575.505,Z 248.605,A 0.000,B 0.000,C 90.000,E1 324.975} C_DIS
LIN {X -0.255,Y -580.599,Z 248.598,A 0.000,B 0.000,C 90.000,E1 323.623} C_DIS
LIN {X 0.258,Y -583.420,Z 248.593,A 0.000,B 0.000,C 90.000,E1 322.763} C_DIS
LIN {X 0.168,Y -587.005,Z 248.587,A 0.000,B 0.000,C 90.000,E1 321.698} C_DIS
LIN {X -0.049,Y -594.299,Z 248.576,A 0.000,B 0.000,C 90.000,E1 319.585} C_DIS
LIN {X 0.148,Y -599.213,Z 248.568,A 0.000,B 0.000,C 90.000,E1 318.243} C_DIS
LIN {X -0.030,Y -604.052,Z 248.561,A 0.000,B 0.000,C 90.000,E1 316.944} C_DIS
LIN {X 0.035,Y -607.851,Z 248.555,A 0.000,B 0.000,C 90.000,E1 315.891} C_DIS
LIN {X 0.338,Y -610.465,Z 248.551,A 0.000,B 0.000,C 90.000,E1 315.081} C_DIS
LIN {X -0.195,Y -612.840,Z 248.546,A 0.000,B 0.000,C 90.000,E1 314.352} C_DIS
LIN {X 0.159,Y -614.940,Z 248.542,A 0.000,B 0.000,C 90.000,E1 313.542} C_DIS
LIN {X 0.112,Y -616.906,Z 248.538,A 0.000,B 0.000,C 90.000,E1 312.771} C_DIS
LIN {X 0.087,Y -618.628,Z 248.533,A 0.000,B 0.000,C 90.000,E1 312.000} C_DIS
LIN {X -0.075,Y -620.570,Z 248.528,A 0.000,B 0.000,C 90.000,E1 310.987} C_DIS
LIN {X 0.253,Y -622.336,Z 248.522,A 0.000,B 0.000,C 90.000,E1 309.930} C_DIS
LIN {X -0.123,Y -623.551,Z 248.518,A 0.000,B 0.000,C 90.000,E1 309.197} C_DIS
LIN {X -0.148,Y -624.937,Z 248.512,A 0.000,B 0.000,C 90.000,E1 308.177} C_DIS
LIN {X -0.155,Y -626.101,Z 248.506,A 0.000,B 0.000,C 90.000,E1 307.156} C_DIS
LIN {X 0.006,Y -626.718,Z 248.502,A 0.000,B 0.000,C 90.000,E1 306.377} C_DIS
LIN {X 0.174,Y -627.122,Z 248.498,A 0.000,B 0.000,C 90.000,E1 305.598} C_DIS
LIN {X -0.181,Y -627.405,Z 248.492,A 0.000,B 0.000,C 90.000,E1 304.612} C_DIS
LIN {X -0.016,Y -627.471,Z 248.487,A 0.000,B 0.000,C 90.000,E1 303.579} C_DIS
LIN {X -0.194,Y -627.341,Z 248.482,A 0.000,B 0.000,C 90.000,E1 302.832} C_DIS
LIN {X -0.039,Y -626.772,Z 248.478,A 0.000,B 0.000,C 90.000,E1 302.054} C_DIS
LIN {X -0.225,Y -625.533,Z 248.472,A 0.000,B 0.000,C 90.000,E1 301.052} C_DIS
LIN {X 0.107,Y -624.478,Z 248.468,A 0.000,B 0.000,C 90.000,E1 300.256} C_DIS
LIN {X -0.113,Y -622.016,Z 248.461,A 0.000,B 0.000,C 90.000,E1 298.999} C_DIS
LIN {X -0.114,Y -620.951,Z 248.458,A 0.000,B 0.000,C 90.000,E1 298.487} C_DIS
LIN {X -0.138,Y -617.822,Z 248.451,A 0.000,B 0.000,C 90.000,E1 297.206} C_DIS
LIN {X 0.061,Y -614.497,Z 248.444,A 0.000,B 0.000,C 90.000,E1 295.899} C_DIS
LIN {X 0.215,Y -610.930,Z 248.437,A 0.000,B 0.000,C 90.000,E1 294.591} C_DIS
LIN {X 0.222,Y -606.240,Z 248.427,A 0.000,B 0.000,C 90.000,E1 292.770} C_DIS
LIN {X -0.124,Y -601.804,Z 248.416,A 0.000,B 0.000,C 90.000,E1 290.972} C_DIS
LIN {X 0.036,Y -596.985,Z 248.405,A 0.000,B 0.000,C 90.000,E1 288.852} C_DIS
LIN {X 0.019,Y -591.369,Z 248.390,A 0.000,B 0.000,C 90.000,E1 286.205} C_DIS
LIN {X 0.116,Y -587.414,Z 248.378,A 0.000,B 0.000,C 90.000,E1 284.064} C_DIS
LIN {X -0.261,Y -583.266,Z 248.363,A 0.000,B 0.000,C 90.000,E1 281.422} C_DIS
LIN {X -0.192,Y -579.781,Z 248.347,A 0.000,B 0.000,C 90.000,E1 278.454} C_DIS
LIN {X -0.208,Y -577.705,Z 248.333,A 0.000,B 0.000,C 90.000,E1 276.024} C_DIS
LIN {X 0.012,Y -576.045,Z 248.315,A 0.000,B 0.000,C 90.000,E1 272.751} C_DIS
LIN {X 0.002,Y -576.243,Z 248.293,A 0.000,B 0.000,C 90.000,E1 268.682} C_DIS
LIN {X 0.111,Y -578.977,Z 248.270,A 0.000,B 0.000,C 90.000,E1 264.609} C_DIS
LIN {X 0.043,Y -581.670,Z 248.257,A 0.000,B 0.000,C 90.000,E1 262.186} C_DIS
LIN {X 0.235,Y -584.925,Z 248.243,A 0.000,B 0.000,C 90.000,E1 259.746} C_DIS
LIN {X -0.191,Y -588.220,Z 248.231,A 0.000,B 0.000,C 90.000,E1 257.645} C_DIS
LIN {X -0.054,Y -590.262,Z 248.224,A 0.000,B 0.000,C 90.000,E1 256.297} C_DIS
LIN {X -0.315,Y -592.300,Z 248.216,A 0.000,B 0.000,C 90.000,E1 254.991} C_DIS
LIN {X 0.067,Y -593.401,Z 248.212,A 0.000,B 0.000,C 90.000,E1 254.157} C_DIS
LIN {X 0.161,Y -594.658,Z 248.206,A 0.000,B 0.000,C 90.000,E1 253.087} C_DIS
LIN {X -0.121,Y -595.555,Z 248.200,A 0.000,B 0.000,C 90.000,E1 252.054} C_DIS
LIN {X 0.181,Y -595.926,Z 248.194,A 0.000,B 0.000,C 90.000,E1 250.967} C_DIS
LIN {X -0.076,Y -596.091,Z 248.189,A 0.000,B 0.000,C 90.000,E1 249.934} C_DIS
LIN {X 0.220,Y -595.989,Z 248.183,A 0.000,B 0.000,C 90.000,E1 248.847} C_DIS
LIN {X -0.289,Y -595.560,Z 248.178,A 0.000,B 0.000,C 90.000,E1 248.103} C_DIS
LIN {X 0.073,Y -595.155,Z 248.175,A 0.000,B 0.000,C 90.000,E1 247.539} C_DIS
LIN {X -0.083,Y -593.592,Z 248.168,A 0.000,B 0.000,C 90.000,E1 246.230} C_DIS
LIN {X 0.172,Y -592.348,Z 248.164,A 0.000,B 0.000,C 90.000,E1 245.409} C_DIS
LIN {X -0.373,Y -590.860,Z 248.159,A 0.000,B 0.000,C 90.000,E1 244.665} C_DIS
LIN {X 0.003,Y -588.612,Z 248.153,A 0.000,B 0.000,C 90.000,E1 243.563} C_DIS
LIN {X 0.084,Y -585.996,Z 248.147,A 0.000,B 0.000,C 90.000,E1 242.487} C_DIS
LIN {X 0.002,Y -584.022,Z 248.143,A 0.000,B 0.000,C 90.000,E1 241.691} C_DIS
LIN {X 0.132,Y -581.940,Z 248.138,A 0.000,B 0.000,C 90.000,E1 240.873} C_DIS
LIN {X 0.157,Y -578.789,Z 248.132,A 0.000,B 0.000,C 90.000,E1 239.793} C_DIS
LIN {X -0.135,Y -577.287,Z 248.129,A 0.000,B 0.000,C 90.000,E1 239.282} C_DIS
LIN {X -0.167,Y -573.783,Z 248.123,A 0.000,B 0.000,C 90.000,E1 238.201} C_DIS
LIN {X 0.009,Y -568.464,Z 248.114,A 0.000,B 0.000,C 90.000,E1 236.548} C_DIS
LIN {X 0.075,Y -563.226,Z 248.105,A 0.000,B 0.000,C 90.000,E1 234.895} C_DIS
LIN {X 0.157,Y -559.835,Z 248.099,A 0.000,B 0.000,C 90.000,E1 233.783} C_DIS
LIN {X 0.235,Y -554.616,Z 248.090,A 0.000,B 0.000,C 90.000,E1 232.110} C_DIS
LIN {X 0.148,Y -550.264,Z 248.082,A 0.000,B 0.000,C 90.000,E1 230.723} C_DIS
LIN {X -0.028,Y -545.892,Z 248.074,A 0.000,B 0.000,C 90.000,E1 229.337} C_DIS
LIN {X 0.020,Y -541.423,Z 248.066,A 0.000,B 0.000,C 90.000,E1 227.919} C_DIS
LIN {X -0.005,Y -535.987,Z 248.057,A 0.000,B 0.000,C 90.000,E1 226.215} C_DIS
LIN {X 0.245,Y -531.445,Z 248.049,A 0.000,B 0.000,C 90.000,E1 224.757} C_DIS
LIN {X -0.062,Y -525.002,Z 248.038,A 0.000,B 0.000,C 90.000,E1 222.771} C_DIS
LIN {X 0.010,Y -520.548,Z 248.030,A 0.000,B 0.000,C 90.000,E1 221.310} C_DIS
LIN {X -0.072,Y -515.317,Z 248.020,A 0.000,B 0.000,C 90.000,E1 219.564} C_DIS
LIN {X -0.284,Y -509.285,Z 248.008,A 0.000,B 0.000,C 90.000,E1 217.523} C_DIS
LIN {X -0.039,Y -505.075,Z 248.000,A 0.000,B 0.000,C 90.000,E1 216.011} C_DIS
LIN {X -0.004,Y -499.135,Z 247.988,A 0.000,B 0.000,C 90.000,E1 213.913} C_DIS
LIN {X 0.011,Y -493.346,Z 247.977,A 0.000,B 0.000,C 90.000,E1 211.799} C_DIS
LIN {X 0.212,Y -489.383,Z 247.968,A 0.000,B 0.000,C 90.000,E1 210.256} C_DIS
LIN {X 0.096,Y -481.975,Z 247.951,A 0.000,B 0.000,C 90.000,E1 207.206} C_DIS
LIN {X -0.252,Y -476.003,Z 247.936,A 0.000,B 0.000,C 90.000,E1 204.463} C_DIS
LIN {X -0.071,Y -471.729,Z 247.924,A 0.000,B 0.000,C 90.000,E1 202.259} C_DIS
LIN {X -0.099,Y -467.928,Z 247.911,A 0.000,B 0.000,C 90.000,E1 200.066} C_DIS
LIN {X 0.151,Y -463.992,Z 247.897,A 0.000,B 0.000,C 90.000,E1 197.511} C_DIS
LIN {X -0.144,Y -460.430,Z 247.883,A 0.000,B 0.000,C 90.000,E1 195.009} C_DIS
LIN {X 0.118,Y -457.951,Z 247.873,A 0.000,B 0.000,C 90.000,E1 193.063} C_DIS
LIN {X 0.001,Y -456.009,Z 247.864,A 0.000,B 0.000,C 90.000,E1 191.478} C_DIS
LIN {X -0.027,Y -453.822,Z 247.853,A 0.000,B 0.000,C 90.000,E1 189.557} C_DIS
LIN {X 0.226,Y -451.164,Z 247.839,A 0.000,B 0.000,C 90.000,E1 186.947} C_DIS
LIN {X -0.214,Y -448.900,Z 247.824,A 0.000,B 0.000,C 90.000,E1 184.416} C_DIS
LIN {X -0.023,Y -447.085,Z 247.812,A 0.000,B 0.000,C 90.000,E1 182.121} C_DIS
LIN {X 0.102,Y -445.564,Z 247.799,A 0.000,B 0.000,C 90.000,E1 179.828} C_DIS
LIN {X -0.126,Y -444.258,Z 247.785,A 0.000,B 0.000,C 90.000,E1 177.249} C_DIS
LIN {X -0.027,Y -443.459,Z 247.767,A 0.000,B 0.000,C 90.000,E1 173.970} C_DIS
LIN {X -0.189,Y -443.395,Z 247.752,A 0.000,B 0.000,C 90.000,E1 171.376} C_DIS
LIN {X -0.060,Y -443.700,Z 247.741,A 0.000,B 0.000,C 90.000,E1 169.398} C_DIS
LIN {X 0.059,Y -444.754,Z 247.723,A 0.000,B 0.000,C 90.000,E1 166.117} C_DIS
LIN {X -0.198,Y -445.484,Z 247.714,A 0.000,B 0.000,C 90.000,E1 164.519} C_DIS
LIN {X -0.171,Y -446.692,Z 247.701,A 0.000,B 0.000,C 90.000,E1 162.236} C_DIS
LIN {X -0.039,Y -449.311,Z 247.681,A 0.000,B 0.000,C 90.000,E1 158.646} C_DIS
LIN {X 0.024,Y -451.798,Z 247.667,A 0.000,B 0.000,C 90.000,E1 156.049} C_DIS
LIN {X 0.200,Y -455.251,Z 247.651,A 0.000,B 0.000,C 90.000,E1 153.127} C_DIS
LIN {X 0.112,Y -459.310,Z 247.635,A 0.000,B 0.000,C 90.000,E1 150.255} C_DIS
LIN {X 0.099,Y -461.724,Z 247.626,A 0.000,B 0.000,C 90.000,E1 148.663} C_DIS
LIN {X -0.018,Y -464.270,Z 247.617,A 0.000,B 0.000,C 90.000,E1 147.089} C_DIS
LIN {X 0.060,Y -467.456,Z 247.607,A 0.000,B 0.000,C 90.000,E1 145.182} C_DIS
LIN {X 0.159,Y -469.473,Z 247.600,A 0.000,B 0.000,C 90.000,E1 143.909} C_DIS
LIN {X 0.131,Y -472.347,Z 247.589,A 0.000,B 0.000,C 90.000,E1 142.029} C_DIS
LIN {X 0.161,Y -474.948,Z 247.579,A 0.000,B 0.000,C 90.000,E1 140.150} C_DIS
LIN {X -0.077,Y -476.464,Z 247.572,A 0.000,B 0.000,C 90.000,E1 138.933} C_DIS
LIN {X 0.030,Y -477.774,Z 247.565,A 0.000,B 0.000,C 90.000,E1 137.676} C_DIS
LIN {X 0.045,Y -478.529,Z 247.560,A 0.000,B 0.000,C 90.000,E1 136.743} C_DIS
LIN {X 0.186,Y -479.337,Z 247.553,A 0.000,B 0.000,C 90.000,E1 135.486} C_DIS
LIN {X -0.008,Y -479.762,Z 247.546,A 0.000,B 0.000,C 90.000,E1 134.271} C_DIS
LIN {X 0.028,Y -479.950,Z 247.541,A 0.000,B 0.000,C 90.000,E1 133.338} C_DIS
LIN {X 0.189,Y -479.658,Z 247.534,A 0.000,B 0.000,C 90.000,E1 132.081} C_DIS
LIN {X 0.022,Y -478.935,Z 247.527,A 0.000,B 0.000,C 90.000,E1 130.862} C_DIS
LIN {X -0.054,Y -477.740,Z 247.518,A 0.000,B 0.000,C 90.000,E1 129.322} C_DIS
LIN {X -0.190,Y -476.579,Z 247.512,A 0.000,B 0.000,C 90.000,E1 128.096} C_DIS
LIN {X 0.042,Y -475.161,Z 247.505,A 0.000,B 0.000,C 90.000,E1 126.824} C_DIS
LIN {X -0.126,Y -473.493,Z 247.498,A 0.000,B 0.000,C 90.000,E1 125.598} C_DIS
LIN {X 0.002,Y -470.625,Z 247.487,A 0.000,B 0.000,C 90.000,E1 123.706} C_DIS
LIN {X 0.187,Y -467.475,Z 247.477,A 0.000,B 0.000,C 90.000,E1 121.799} C_DIS
LIN {X 0.049,Y -464.178,Z 247.466,A 0.000,B 0.000,C 90.000,E1 119.922} C_DIS
LIN {X -0.124,Y -461.373,Z 247.458,A 0.000,B 0.000,C 90.000,E1 118.359} C_DIS
LIN {X -0.034,Y -457.918,Z 247.447,A 0.000,B 0.000,C 90.000,E1 116.437} C_DIS
LIN {X -0.026,Y -454.482,Z 247.436,A 0.000,B 0.000,C 90.000,E1 114.515} C_DIS
LIN {X 0.144,Y -450.684,Z 247.424,A 0.000,B 0.000,C 90.000,E1 112.280} C_DIS
LIN {X 0.104,Y -450.677,Z 247.424,A 0.000,B 0.000,C 90.000,E1 112.280} C_DIS
LIN {X 0.072,Y -456.719,Z 247.411,A 0.000,B 0.000,C 90.000,E1 109.993} C_DIS
LIN {X -0.028,Y -457.503,Z 247.409,A 0.000,B 0.000,C 90.000,E1 109.685} C_DIS
LIN {X -0.083,Y -466.179,Z 247.386,A 0.000,B 0.000,C 90.000,E1 105.552} C_DIS
LIN {X 0.094,Y -467.746,Z 247.383,A 0.000,B 0.000,C 90.000,E1 104.898} C_DIS
LIN {X 0.066,Y -475.953,Z 247.357,A 0.000,B 0.000,C 90.000,E1 100.197} C_DIS
LIN {X 0.216,Y -476.672,Z 247.353,A 0.000,B 0.000,C 90.000,E1 99.557} C_DIS
LIN {X -0.140,Y -481.903,Z 247.331,A 0.000,B 0.000,C 90.000,E1 95.568} C_DIS
LIN {X 0.188,Y -482.200,Z 247.329,A 0.000,B 0.000,C 90.000,E1 95.220} C_DIS
LIN {X 0.127,Y -485.383,Z 247.305,A 0.000,B 0.000,C 90.000,E1 90.917} C_DIS
LIN {X -0.049,Y -485.530,Z 247.304,A 0.000,B 0.000,C 90.000,E1 90.630} C_DIS
LIN {X 0.160,Y -486.354,Z 247.281,A 0.000,B 0.000,C 90.000,E1 86.617} C_DIS
LIN {X -0.016,Y -486.369,Z 247.280,A 0.000,B 0.000,C 90.000,E1 86.331} C_DIS
LIN {X -0.027,Y -485.862,Z 247.275,A 0.000,B 0.000,C 90.000,E1 85.412} C_DIS
LIN {X 0.008,Y -484.692,Z 247.254,A 0.000,B 0.000,C 90.000,E1 81.724} C_DIS
LIN {X -0.125,Y -484.513,Z 247.252,A 0.000,B 0.000,C 90.000,E1 81.432} C_DIS
LIN {X -0.254,Y -480.448,Z 247.227,A 0.000,B 0.000,C 90.000,E1 76.825} C_DIS
LIN {X 0.095,Y -474.214,Z 247.201,A 0.000,B 0.000,C 90.000,E1 72.127} C_DIS
LIN {X 0.029,Y -473.061,Z 247.197,A 0.000,B 0.000,C 90.000,E1 71.511} C_DIS
LIN {X 0.044,Y -465.481,Z 247.172,A 0.000,B 0.000,C 90.000,E1 66.975} C_DIS
LIN {X 0.004,Y -465.472,Z 247.172,A 0.000,B 0.000,C 90.000,E1 66.975} C_DIS
LIN {X -0.033,Y -469.941,Z 247.162,A 0.000,B 0.000,C 90.000,E1 65.229} C_DIS
LIN {X -0.026,Y -473.171,Z 247.155,A 0.000,B 0.000,C 90.000,E1 63.973} C_DIS
LIN {X -0.041,Y -478.100,Z 247.145,A 0.000,B 0.000,C 90.000,E1 62.103} C_DIS
LIN {X 0.087,Y -483.941,Z 247.133,A 0.000,B 0.000,C 90.000,E1 59.921} C_DIS
LIN {X -0.106,Y -488.180,Z 247.124,A 0.000,B 0.000,C 90.000,E1 58.408} C_DIS
LIN {X 0.040,Y -491.576,Z 247.118,A 0.000,B 0.000,C 90.000,E1 57.168} C_DIS
LIN {X -0.032,Y -494.846,Z 247.111,A 0.000,B 0.000,C 90.000,E1 55.960} C_DIS
LIN {X -0.195,Y -497.939,Z 247.104,A 0.000,B 0.000,C 90.000,E1 54.769} C_DIS
LIN {X -0.016,Y -500.802,Z 247.098,A 0.000,B 0.000,C 90.000,E1 53.543} C_DIS
LIN {X 0.024,Y -502.884,Z 247.092,A 0.000,B 0.000,C 90.000,E1 52.637} C_DIS
LIN {X -0.007,Y -504.818,Z 247.088,A 0.000,B 0.000,C 90.000,E1 51.743} C_DIS
LIN {X -0.114,Y -507.073,Z 247.081,A 0.000,B 0.000,C 90.000,E1 50.561} C_DIS
LIN {X -0.192,Y -509.150,Z 247.074,A 0.000,B 0.000,C 90.000,E1 49.380} C_DIS
LIN {X 0.090,Y -510.924,Z 247.068,A 0.000,B 0.000,C 90.000,E1 48.162} C_DIS
LIN {X -0.233,Y -512.019,Z 247.063,A 0.000,B 0.000,C 90.000,E1 47.310} C_DIS
LIN {X 0.179,Y -512.931,Z 247.058,A 0.000,B 0.000,C 90.000,E1 46.377} C_DIS
LIN {X -0.031,Y -513.503,Z 247.055,A 0.000,B 0.000,C 90.000,E1 45.810} C_DIS
LIN {X 0.292,Y -514.250,Z 247.048,A 0.000,B 0.000,C 90.000,E1 44.595} C_DIS
LIN {X 0.002,Y -514.655,Z 247.043,A 0.000,B 0.000,C 90.000,E1 43.743} C_DIS
LIN {X 0.339,Y -514.959,Z 247.037,A 0.000,B 0.000,C 90.000,E1 42.528} C_DIS
LIN {X 0.057,Y -515.028,Z 247.032,A 0.000,B 0.000,C 90.000,E1 41.676} C_DIS
LIN {X 0.164,Y -514.901,Z 247.027,A 0.000,B 0.000,C 90.000,E1 40.782} C_DIS
LIN {X -0.121,Y -514.569,Z 247.022,A 0.000,B 0.000,C 90.000,E1 39.930} C_DIS
LIN {X -0.171,Y -513.653,Z 247.014,A 0.000,B 0.000,C 90.000,E1 38.463} C_DIS
LIN {X -0.083,Y -512.888,Z 247.009,A 0.000,B 0.000,C 90.000,E1 37.569} C_DIS
LIN {X 0.012,Y -511.559,Z 247.002,A 0.000,B 0.000,C 90.000,E1 36.377} C_DIS
LIN {X -0.236,Y -510.340,Z 246.997,A 0.000,B 0.000,C 90.000,E1 35.518} C_DIS
LIN {X 0.151,Y -508.152,Z 246.989,A 0.000,B 0.000,C 90.000,E1 33.992} C_DIS
LIN {X -0.207,Y -505.826,Z 246.981,A 0.000,B 0.000,C 90.000,E1 32.546} C_DIS
LIN {X 0.121,Y -503.096,Z 246.971,A 0.000,B 0.000,C 90.000,E1 30.718} C_DIS
LIN {X -0.216,Y -499.743,Z 246.957,A 0.000,B 0.000,C 90.000,E1 28.359} C_DIS
LIN {X 0.074,Y -497.923,Z 246.949,A 0.000,B 0.000,C 90.000,E1 26.821} C_DIS
LIN {X 0.243,Y -495.286,Z 246.936,A 0.000,B 0.000,C 90.000,E1 24.387} C_DIS
LIN {X 0.125,Y -493.204,Z 246.924,A 0.000,B 0.000,C 90.000,E1 22.280} C_DIS
LIN {X -0.083,Y -491.530,Z 246.914,A 0.000,B 0.000,C 90.000,E1 20.482} C_DIS
LIN {X -0.181,Y -489.732,Z 246.902,A 0.000,B 0.000,C 90.000,E1 18.362} C_DIS
LIN {X 0.117,Y -488.268,Z 246.892,A 0.000,B 0.000,C 90.000,E1 16.496} C_DIS
LIN {X 0.109,Y -486.702,Z 246.880,A 0.000,B 0.000,C 90.000,E1 14.356} C_DIS
LIN {X 0.181,Y -485.236,Z 246.866,A 0.000,B 0.000,C 90.000,E1 11.895} C_DIS
LIN {X 0.127,Y -484.238,Z 246.853,A 0.000,B 0.000,C 90.000,E1 9.443} C_DIS
LIN {X 0.083,Y -483.601,Z 246.841,A 0.000,B 0.000,C 90.000,E1 7.296} C_DIS
LIN {X 0.037,Y -483.220,Z 246.825,A 0.000,B 0.000,C 90.000,E1 4.531} C_DIS
LIN {X -0.237,Y -483.342,Z 246.813,A 0.000,B 0.000,C 90.000,E1 2.407} C_DIS
LIN {X -0.174,Y -484.229,Z 246.795,A 0.000,B 0.000,C 90.000,E1 359.198} C_DIS
LIN {X 0.205,Y -485.993,Z 246.780,A 0.000,B 0.000,C 90.000,E1 356.388} C_DIS
LIN {X 0.183,Y -487.430,Z 246.770,A 0.000,B 0.000,C 90.000,E1 354.552} C_DIS
LIN {X -0.165,Y -492.074,Z 246.748,A 0.000,B 0.000,C 90.000,E1 350.622} C_DIS
LIN {X 0.206,Y -495.508,Z 246.738,A 0.000,B 0.000,C 90.000,E1 348.757} C_DIS
LIN {X -0.030,Y -504.918,Z 246.718,A 0.000,B 0.000,C 90.000,E1 345.172} C_DIS
LIN {X -0.063,Y -509.015,Z 246.709,A 0.000,B 0.000,C 90.000,E1 343.685} C_DIS
LIN {X 0.195,Y -514.756,Z 246.698,A 0.000,B 0.000,C 90.000,E1 341.583} C_DIS
LIN {X -0.269,Y -524.694,Z 246.680,A 0.000,B 0.000,C 90.000,E1 338.411} C_DIS
LIN {X -0.212,Y -530.629,Z 246.670,A 0.000,B 0.000,C 90.000,E1 336.666} C_DIS
LIN {X -0.022,Y -536.661,Z 246.661,A 0.000,B 0.000,C 90.000,E1 334.921} C_DIS
LIN {X 0.245,Y -544.937,Z 246.648,A 0.000,B 0.000,C 90.000,E1 332.615} C_DIS
LIN {X -0.258,Y -550.273,Z 246.640,A 0.000,B 0.000,C 90.000,E1 331.257} C_DIS
LIN {X 0.072,Y -555.514,Z 246.632,A 0.000,B 0.000,C 90.000,E1 329.822} C_DIS
LIN {X -0.177,Y -560.543,Z 246.625,A 0.000,B 0.000,C 90.000,E1 328.456} C_DIS
LIN {X 0.166,Y -568.616,Z 246.612,A 0.000,B 0.000,C 90.000,E1 326.215} C_DIS
LIN {X -0.175,Y -574.930,Z 246.603,A 0.000,B 0.000,C 90.000,E1 324.609} C_DIS
LIN {X 0.090,Y -578.997,Z 246.597,A 0.000,B 0.000,C 90.000,E1 323.497} C_DIS
LIN {X 0.121,Y -581.805,Z 246.593,A 0.000,B 0.000,C 90.000,E1 322.683} C_DIS
LIN {X 0.193,Y -586.249,Z 246.585,A 0.000,B 0.000,C 90.000,E1 321.331} C_DIS
LIN {X 0.149,Y -596.826,Z 246.569,A 0.000,B 0.000,C 90.000,E1 318.405} C_DIS
LIN {X -0.071,Y -601.793,Z 246.562,A 0.000,B 0.000,C 90.000,E1 317.106} C_DIS
LIN {X -0.237,Y -606.573,Z 246.554,A 0.000,B 0.000,C 90.000,E1 315.810} C_DIS
LIN {X 0.052,Y -609.149,Z 246.550,A 0.000,B 0.000,C 90.000,E1 315.000} C_DIS
LIN {X 0.370,Y -611.543,Z 246.546,A 0.000,B 0.000,C 90.000,E1 314.190} C_DIS
LIN {X -0.156,Y -613.612,Z 246.541,A 0.000,B 0.000,C 90.000,E1 313.461} C_DIS
LIN {X 0.069,Y -616.138,Z 246.536,A 0.000,B 0.000,C 90.000,E1 312.405} C_DIS
LIN {X -0.282,Y -618.621,Z 246.529,A 0.000,B 0.000,C 90.000,E1 311.148} C_DIS
LIN {X 0.180,Y -619.980,Z 246.524,A 0.000,B 0.000,C 90.000,E1 310.334} C_DIS
LIN {X 0.180,Y -621.222,Z 246.520,A 0.000,B 0.000,C 90.000,E1 309.564} C_DIS
LIN {X -0.205,Y -622.330,Z 246.516,A 0.000,B 0.000,C 90.000,E1 308.830} C_DIS
LIN {X -0.247,Y -623.581,Z 246.510,A 0.000,B 0.000,C 90.000,E1 307.810} C_DIS
LIN {X -0.073,Y -624.171,Z 246.507,A 0.000,B 0.000,C 90.000,E1 307.282} C_DIS
LIN {X 0.063,Y -624.795,Z 246.503,A 0.000,B 0.000,C 90.000,E1 306.503} C_DIS
LIN {X -0.324,Y -625.307,Z 246.497,A 0.000,B 0.000,C 90.000,E1 305.518} C_DIS
LIN {X -0.190,Y -625.579,Z 246.492,A 0.000,B 0.000,C 90.000,E1 304.485} C_DIS
LIN {X -0.047,Y -625.632,Z 246.486,A 0.000,B 0.000,C 90.000,E1 303.452} C_DIS
LIN {X -0.238,Y -625.522,Z 246.483,A 0.000,B 0.000,C 90.000,E1 302.959} C_DIS
LIN {X 0.094,Y -625.052,Z 246.479,A 0.000,B 0.000,C 90.000,E1 302.163} C_DIS
LIN {X 0.220,Y -623.554,Z 246.472,A 0.000,B 0.000,C 90.000,E1 300.875} C_DIS
LIN {X 0.001,Y -622.825,Z 246.469,A 0.000,B 0.000,C 90.000,E1 300.384} C_DIS
LIN {X 0.295,Y -620.416,Z 246.462,A 0.000,B 0.000,C 90.000,E1 299.077} C_DIS
LIN {X -0.269,Y -618.756,Z 246.457,A 0.000,B 0.000,C 90.000,E1 298.359} C_DIS
LIN {X -0.046,Y -615.677,Z 246.450,A 0.000,B 0.000,C 90.000,E1 297.052} C_DIS
LIN {X -0.165,Y -612.318,Z 246.443,A 0.000,B 0.000,C 90.000,E1 295.771} C_DIS
LIN {X 0.319,Y -606.037,Z 246.430,A 0.000,B 0.000,C 90.000,E1 293.387} C_DIS
LIN {X 0.153,Y -600.275,Z 246.417,A 0.000,B 0.000,C 90.000,E1 291.046} C_DIS
LIN {X -0.089,Y -595.456,Z 246.405,A 0.000,B 0.000,C 90.000,E1 288.960} C_DIS
LIN {X -0.173,Y -589.843,Z 246.391,A 0.000,B 0.000,C 90.000,E1 286.315} C_DIS
LIN {X -0.202,Y -586.826,Z 246.382,A 0.000,B 0.000,C 90.000,E1 284.717} C_DIS
LIN {X -0.232,Y -582.076,Z 246.365,A 0.000,B 0.000,C 90.000,E1 281.771} C_DIS
LIN {X -0.214,Y -578.458,Z 246.349,A 0.000,B 0.000,C 90.000,E1 278.803} C_DIS
LIN {X 0.069,Y -575.866,Z 246.332,A 0.000,B 0.000,C 90.000,E1 275.796} C_DIS
LIN {X 0.253,Y -574.176,Z 246.302,A 0.000,B 0.000,C 90.000,E1 270.344} C_DIS
LIN {X 0.238,Y -576.736,Z 246.273,A 0.000,B 0.000,C 90.000,E1 265.184} C_DIS
LIN {X 0.099,Y -579.311,Z 246.260,A 0.000,B 0.000,C 90.000,E1 262.761} C_DIS
LIN {X 0.128,Y -582.414,Z 246.246,A 0.000,B 0.000,C 90.000,E1 260.330} C_DIS
LIN {X 0.204,Y -585.669,Z 246.234,A 0.000,B 0.000,C 90.000,E1 258.173} C_DIS
LIN {X -0.021,Y -588.165,Z 246.226,A 0.000,B 0.000,C 90.000,E1 256.589} C_DIS
LIN {X -0.056,Y -590.605,Z 246.217,A 0.000,B 0.000,C 90.000,E1 254.991} C_DIS
LIN {X 0.308,Y -591.723,Z 246.212,A 0.000,B 0.000,C 90.000,E1 254.157} C_DIS
LIN {X -0.189,Y -593.007,Z 246.206,A 0.000,B 0.000,C 90.000,E1 253.142} C_DIS
LIN {X 0.074,Y -593.917,Z 246.200,A 0.000,B 0.000,C 90.000,E1 252.054} C_DIS
LIN {X 0.160,Y -594.280,Z 246.195,A 0.000,B 0.000,C 90.000,E1 250.986} C_DIS
LIN {X 0.182,Y -594.443,Z 246.190,A 0.000,B 0.000,C 90.000,E1 250.188} C_DIS
LIN {X 0.108,Y -594.391,Z 246.184,A 0.000,B 0.000,C 90.000,E1 249.135} C_DIS
LIN {X 0.244,Y -594.221,Z 246.181,A 0.000,B 0.000,C 90.000,E1 248.592} C_DIS
LIN {X 0.172,Y -593.540,Z 246.175,A 0.000,B 0.000,C 90.000,E1 247.539} C_DIS
LIN {X -0.012,Y -591.976,Z 246.168,A 0.000,B 0.000,C 90.000,E1 246.230} C_DIS
LIN {X 0.226,Y -590.737,Z 246.164,A 0.000,B 0.000,C 90.000,E1 245.409} C_DIS
LIN {X -0.335,Y -589.239,Z 246.159,A 0.000,B 0.000,C 90.000,E1 244.665} C_DIS
LIN {X -0.131,Y -587.583,Z 246.155,A 0.000,B 0.000,C 90.000,E1 243.845} C_DIS
LIN {X 0.314,Y -585.718,Z 246.150,A 0.000,B 0.000,C 90.000,E1 242.999} C_DIS
LIN {X -0.023,Y -582.387,Z 246.143,A 0.000,B 0.000,C 90.000,E1 241.691} C_DIS
LIN {X 0.090,Y -580.264,Z 246.138,A 0.000,B 0.000,C 90.000,E1 240.873} C_DIS
LIN {X -0.057,Y -576.357,Z 246.131,A 0.000,B 0.000,C 90.000,E1 239.537} C_DIS
LIN {X -0.265,Y -572.114,Z 246.123,A 0.000,B 0.000,C 90.000,E1 238.201} C_DIS
LIN {X -0.244,Y -567.644,Z 246.116,A 0.000,B 0.000,C 90.000,E1 236.834} C_DIS
LIN {X -0.196,Y -562.412,Z 246.107,A 0.000,B 0.000,C 90.000,E1 235.182} C_DIS
LIN {X -0.124,Y -559.017,Z 246.100,A 0.000,B 0.000,C 90.000,E1 234.069} C_DIS
LIN {X -0.063,Y -553.746,Z 246.091,A 0.000,B 0.000,C 90.000,E1 232.396} C_DIS
LIN {X -0.162,Y -549.392,Z 246.083,A 0.000,B 0.000,C 90.000,E1 231.009} C_DIS
LIN {X 0.009,Y -544.987,Z 246.076,A 0.000,B 0.000,C 90.000,E1 229.585} C_DIS
LIN {X 0.108,Y -539.621,Z 246.066,A 0.000,B 0.000,C 90.000,E1 227.877} C_DIS
LIN {X 0.016,Y -534.169,Z 246.057,A 0.000,B 0.000,C 90.000,E1 226.176} C_DIS
LIN {X -0.134,Y -529.585,Z 246.049,A 0.000,B 0.000,C 90.000,E1 224.757} C_DIS
LIN {X -0.051,Y -524.054,Z 246.039,A 0.000,B 0.000,C 90.000,E1 223.014} C_DIS
LIN {X 0.291,Y -518.695,Z 246.029,A 0.000,B 0.000,C 90.000,E1 221.229} C_DIS
LIN {X 0.165,Y -513.445,Z 246.020,A 0.000,B 0.000,C 90.000,E1 219.483} C_DIS
LIN {X -0.100,Y -507.431,Z 246.008,A 0.000,B 0.000,C 90.000,E1 217.443} C_DIS
LIN {X 0.213,Y -504.074,Z 246.001,A 0.000,B 0.000,C 90.000,E1 216.217} C_DIS
LIN {X 0.217,Y -498.120,Z 245.990,A 0.000,B 0.000,C 90.000,E1 214.119} C_DIS
LIN {X 0.204,Y -492.288,Z 245.978,A 0.000,B 0.000,C 90.000,E1 212.005} C_DIS
LIN {X -0.036,Y -488.279,Z 245.970,A 0.000,B 0.000,C 90.000,E1 210.512} C_DIS
LIN {X 0.027,Y -482.164,Z 245.956,A 0.000,B 0.000,C 90.000,E1 208.052} C_DIS
LIN {X -0.080,Y -476.691,Z 245.942,A 0.000,B 0.000,C 90.000,E1 205.591} C_DIS
LIN {X 0.123,Y -472.269,Z 245.930,A 0.000,B 0.000,C 90.000,E1 203.387} C_DIS
LIN {X 0.067,Y -466.105,Z 245.911,A 0.000,B 0.000,C 90.000,E1 199.939} C_DIS
LIN {X 0.035,Y -461.744,Z 245.895,A 0.000,B 0.000,C 90.000,E1 197.094} C_DIS
LIN {X -0.102,Y -457.872,Z 245.879,A 0.000,B 0.000,C 90.000,E1 194.245} C_DIS
LIN {X -0.126,Y -455.091,Z 245.867,A 0.000,B 0.000,C 90.000,E1 192.007} C_DIS
LIN {X -0.124,Y -452.076,Z 245.852,A 0.000,B 0.000,C 90.000,E1 189.434} C_DIS
LIN {X -0.188,Y -449.771,Z 245.840,A 0.000,B 0.000,C 90.000,E1 187.182} C_DIS
LIN {X 0.095,Y -447.721,Z 245.827,A 0.000,B 0.000,C 90.000,E1 184.878} C_DIS
LIN {X 0.140,Y -446.147,Z 245.816,A 0.000,B 0.000,C 90.000,E1 182.922} C_DIS
LIN {X -0.214,Y -444.508,Z 245.804,A 0.000,B 0.000,C 90.000,E1 180.688} C_DIS
LIN {X -0.027,Y -443.010,Z 245.789,A 0.000,B 0.000,C 90.000,E1 178.051} C_DIS
LIN {X -0.043,Y -442.016,Z 245.771,A 0.000,B 0.000,C 90.000,E1 174.780} C_DIS
LIN {X 0.065,Y -441.836,Z 245.753,A 0.000,B 0.000,C 90.000,E1 171.489} C_DIS
LIN {X 0.162,Y -442.138,Z 245.742,A 0.000,B 0.000,C 90.000,E1 169.511} C_DIS
LIN {X 0.230,Y -443.179,Z 245.724,A 0.000,B 0.000,C 90.000,E1 166.228} C_DIS
LIN {X -0.049,Y -443.975,Z 245.715,A 0.000,B 0.000,C 90.000,E1 164.629} C_DIS
LIN {X 0.089,Y -445.311,Z 245.700,A 0.000,B 0.000,C 90.000,E1 162.000} C_DIS
LIN {X -0.135,Y -447.657,Z 245.682,A 0.000,B 0.000,C 90.000,E1 158.773} C_DIS
LIN {X 0.117,Y -449.480,Z 245.671,A 0.000,B 0.000,C 90.000,E1 156.794} C_DIS
LIN {X 0.059,Y -451.977,Z 245.659,A 0.000,B 0.000,C 90.000,E1 154.537} C_DIS
LIN {X -0.060,Y -455.309,Z 245.644,A 0.000,B 0.000,C 90.000,E1 151.975} C_DIS
LIN {X -0.045,Y -458.114,Z 245.634,A 0.000,B 0.000,C 90.000,E1 150.049} C_DIS
LIN {X 0.169,Y -461.605,Z 245.621,A 0.000,B 0.000,C 90.000,E1 147.788} C_DIS
LIN {X 0.074,Y -465.806,Z 245.607,A 0.000,B 0.000,C 90.000,E1 145.261} C_DIS
LIN {X -0.090,Y -468.347,Z 245.598,A 0.000,B 0.000,C 90.000,E1 143.703} C_DIS
LIN {X 0.078,Y -470.727,Z 245.590,A 0.000,B 0.000,C 90.000,E1 142.110} C_DIS
LIN {X 0.067,Y -473.331,Z 245.579,A 0.000,B 0.000,C 90.000,E1 140.231} C_DIS
LIN {X -0.195,Y -474.884,Z 245.572,A 0.000,B 0.000,C 90.000,E1 139.013} C_DIS
LIN {X -0.115,Y -476.173,Z 245.565,A 0.000,B 0.000,C 90.000,E1 137.757} C_DIS
LIN {X -0.118,Y -476.959,Z 245.560,A 0.000,B 0.000,C 90.000,E1 136.824} C_DIS
LIN {X -0.002,Y -477.736,Z 245.553,A 0.000,B 0.000,C 90.000,E1 135.567} C_DIS
LIN {X -0.219,Y -478.213,Z 245.546,A 0.000,B 0.000,C 90.000,E1 134.352} C_DIS
LIN {X 0.127,Y -478.345,Z 245.541,A 0.000,B 0.000,C 90.000,E1 133.380} C_DIS
LIN {X -0.065,Y -478.107,Z 245.534,A 0.000,B 0.000,C 90.000,E1 132.162} C_DIS
LIN {X -0.047,Y -477.624,Z 245.529,A 0.000,B 0.000,C 90.000,E1 131.229} C_DIS
LIN {X -0.041,Y -476.986,Z 245.524,A 0.000,B 0.000,C 90.000,E1 130.297} C_DIS
LIN {X 0.110,Y -476.042,Z 245.517,A 0.000,B 0.000,C 90.000,E1 129.036} C_DIS
LIN {X -0.050,Y -474.858,Z 245.510,A 0.000,B 0.000,C 90.000,E1 127.810} C_DIS
LIN {X -0.222,Y -473.396,Z 245.503,A 0.000,B 0.000,C 90.000,E1 126.583} C_DIS
LIN {X 0.178,Y -472.177,Z 245.498,A 0.000,B 0.000,C 90.000,E1 125.598} C_DIS
LIN {X 0.273,Y -469.297,Z 245.487,A 0.000,B 0.000,C 90.000,E1 123.706} C_DIS
LIN {X 0.274,Y -466.714,Z 245.479,A 0.000,B 0.000,C 90.000,E1 122.133} C_DIS
LIN {X -0.166,Y -464.525,Z 245.472,A 0.000,B 0.000,C 90.000,E1 120.924} C_DIS
LIN {X -0.238,Y -462.347,Z 245.465,A 0.000,B 0.000,C 90.000,E1 119.667} C_DIS
LIN {X 0.086,Y -458.954,Z 245.454,A 0.000,B 0.000,C 90.000,E1 117.719} C_DIS
LIN {X 0.122,Y -455.501,Z 245.443,A 0.000,B 0.000,C 90.000,E1 115.796} C_DIS
LIN {X -0.045,Y -451.540,Z 245.431,A 0.000,B 0.000,C 90.000,E1 113.567} C_DIS
LIN {X -0.228,Y -449.927,Z 245.426,A 0.000,B 0.000,C 90.000,E1 112.642} C_DIS
LIN {X 0.149,Y -449.918,Z 245.426,A 0.000,B 0.000,C 90.000,E1 112.589} C_DIS
LIN {X 0.154,Y -456.689,Z 245.411,A 0.000,B 0.000,C 90.000,E1 109.993} C_DIS
LIN {X 0.054,Y -457.484,Z 245.409,A 0.000,B 0.000,C 90.000,E1 109.685} C_DIS
LIN {X 0.000,Y -466.155,Z 245.386,A 0.000,B 0.000,C 90.000,E1 105.552} C_DIS
LIN {X 0.176,Y -467.723,Z 245.383,A 0.000,B 0.000,C 90.000,E1 104.898} C_DIS
LIN {X 0.150,Y -475.931,Z 245.357,A 0.000,B 0.000,C 90.000,E1 100.197} C_DIS
LIN {X -0.011,Y -476.363,Z 245.355,A 0.000,B 0.000,C 90.000,E1 99.905} C_DIS
LIN {X -0.056,Y -481.887,Z 245.331,A 0.000,B 0.000,C 90.000,E1 95.568} C_DIS
LIN {X -0.208,Y -482.196,Z 245.329,A 0.000,B 0.000,C 90.000,E1 95.277} C_DIS
LIN {X 0.211,Y -485.372,Z 245.305,A 0.000,B 0.000,C 90.000,E1 90.917} C_DIS
LIN {X 0.035,Y -485.531,Z 245.304,A 0.000,B 0.000,C 90.000,E1 90.630} C_DIS
LIN {X 0.243,Y -486.349,Z 245.281,A 0.000,B 0.000,C 90.000,E1 86.617} C_DIS
LIN {X 0.068,Y -486.370,Z 245.280,A 0.000,B 0.000,C 90.000,E1 86.331} C_DIS
LIN {X 0.235,Y -486.058,Z 245.276,A 0.000,B 0.000,C 90.000,E1 85.698} C_DIS
LIN {X 0.092,Y -484.693,Z 245.254,A 0.000,B 0.000,C 90.000,E1 81.724} C_DIS
LIN {X -0.041,Y -484.525,Z 245.252,A 0.000,B 0.000,C 90.000,E1 81.432} C_DIS
LIN {X -0.170,Y -480.462,Z 245.227,A 0.000,B 0.000,C 90.000,E1 76.825} C_DIS
LIN {X 0.178,Y -474.224,Z 245.201,A 0.000,B 0.000,C 90.000,E1 72.127} C_DIS
LIN {X 0.145,Y -473.720,Z 245.199,A 0.000,B 0.000,C 90.000,E1 71.819} C_DIS
LIN {X 0.088,Y -466.169,Z 245.175,A 0.000,B 0.000,C 90.000,E1 67.433} C_DIS
LIN {X 0.210,Y -465.743,Z 245.173,A 0.000,B 0.000,C 90.000,E1 67.102} C_DIS
LIN {X -0.263,Y -464.842,Z 245.171,A 0.000,B 0.000,C 90.000,E1 66.741} C_DIS
LIN {X -0.119,Y -464.844,Z 245.171,A 0.000,B 0.000,C 90.000,E1 66.719} C_DIS
LIN {X 0.032,Y -468.596,Z 245.162,A 0.000,B 0.000,C 90.000,E1 65.229} C_DIS
LIN {X 0.018,Y -471.809,Z 245.155,A 0.000,B 0.000,C 90.000,E1 63.973} C_DIS
LIN {X -0.026,Y -476.779,Z 245.145,A 0.000,B 0.000,C 90.000,E1 62.103} C_DIS
LIN {X 0.065,Y -482.598,Z 245.133,A 0.000,B 0.000,C 90.000,E1 59.921} C_DIS
LIN {X 0.079,Y -487.644,Z 245.123,A 0.000,B 0.000,C 90.000,E1 58.074} C_DIS
LIN {X 0.055,Y -491.853,Z 245.114,A 0.000,B 0.000,C 90.000,E1 56.548} C_DIS
LIN {X -0.164,Y -495.795,Z 245.106,A 0.000,B 0.000,C 90.000,E1 55.055} C_DIS
LIN {X -0.020,Y -498.701,Z 245.099,A 0.000,B 0.000,C 90.000,E1 53.829} C_DIS
LIN {X -0.127,Y -501.473,Z 245.092,A 0.000,B 0.000,C 90.000,E1 52.637} C_DIS
LIN {X 0.106,Y -503.926,Z 245.086,A 0.000,B 0.000,C 90.000,E1 51.412} C_DIS
LIN {X 0.087,Y -505.595,Z 245.081,A 0.000,B 0.000,C 90.000,E1 50.517} C_DIS
LIN {X 0.208,Y -508.132,Z 245.072,A 0.000,B 0.000,C 90.000,E1 49.013} C_DIS
LIN {X 0.093,Y -509.757,Z 245.066,A 0.000,B 0.000,C 90.000,E1 47.838} C_DIS
LIN {X 0.134,Y -510.808,Z 245.061,A 0.000,B 0.000,C 90.000,E1 46.944} C_DIS
LIN {X -0.313,Y -511.903,Z 245.054,A 0.000,B 0.000,C 90.000,E1 45.810} C_DIS
LIN {X -0.015,Y -512.699,Z 245.048,A 0.000,B 0.000,C 90.000,E1 44.595} C_DIS
LIN {X 0.034,Y -513.144,Z 245.043,A 0.000,B 0.000,C 90.000,E1 43.704} C_DIS
LIN {X -0.009,Y -513.401,Z 245.036,A 0.000,B 0.000,C 90.000,E1 42.528} C_DIS
LIN {X 0.078,Y -513.424,Z 245.031,A 0.000,B 0.000,C 90.000,E1 41.634} C_DIS
LIN {X -0.217,Y -513.231,Z 245.026,A 0.000,B 0.000,C 90.000,E1 40.782} C_DIS
LIN {X 0.121,Y -512.730,Z 245.020,A 0.000,B 0.000,C 90.000,E1 39.564} C_DIS
LIN {X 0.120,Y -511.997,Z 245.013,A 0.000,B 0.000,C 90.000,E1 38.382} C_DIS
LIN {X 0.016,Y -510.477,Z 245.005,A 0.000,B 0.000,C 90.000,E1 36.916} C_DIS
LIN {X 0.074,Y -508.927,Z 244.999,A 0.000,B 0.000,C 90.000,E1 35.724} C_DIS
LIN {X 0.013,Y -506.713,Z 244.990,A 0.000,B 0.000,C 90.000,E1 34.246} C_DIS
LIN {X -0.159,Y -505.339,Z 244.985,A 0.000,B 0.000,C 90.000,E1 33.372} C_DIS
LIN {X -0.142,Y -502.905,Z 244.977,A 0.000,B 0.000,C 90.000,E1 31.878} C_DIS
LIN {X 0.161,Y -499.712,Z 244.965,A 0.000,B 0.000,C 90.000,E1 29.745} C_DIS
LIN {X 0.243,Y -497.662,Z 244.957,A 0.000,B 0.000,C 90.000,E1 28.231} C_DIS
LIN {X -0.085,Y -495.143,Z 244.945,A 0.000,B 0.000,C 90.000,E1 26.155} C_DIS
LIN {X -0.015,Y -492.979,Z 244.934,A 0.000,B 0.000,C 90.000,E1 24.027} C_DIS
LIN {X 0.004,Y -490.974,Z 244.922,A 0.000,B 0.000,C 90.000,E1 21.897} C_DIS
LIN {X 0.027,Y -489.292,Z 244.912,A 0.000,B 0.000,C 90.000,E1 20.066} C_DIS
LIN {X 0.012,Y -487.810,Z 244.901,A 0.000,B 0.000,C 90.000,E1 18.236} C_DIS
LIN {X 0.122,Y -486.331,Z 244.891,A 0.000,B 0.000,C 90.000,E1 16.386} C_DIS
LIN {X 0.074,Y -484.798,Z 244.879,A 0.000,B 0.000,C 90.000,E1 14.245} C_DIS
LIN {X -0.144,Y -483.535,Z 244.867,A 0.000,B 0.000,C 90.000,E1 12.119} C_DIS
LIN {X 0.210,Y -482.470,Z 244.854,A 0.000,B 0.000,C 90.000,E1 9.613} C_DIS
LIN {X -0.221,Y -481.924,Z 244.843,A 0.000,B 0.000,C 90.000,E1 7.814} C_DIS
LIN {X 0.153,Y -481.374,Z 244.828,A 0.000,B 0.000,C 90.000,E1 4.992} C_DIS
LIN {X 0.153,Y -481.444,Z 244.814,A 0.000,B 0.000,C 90.000,E1 2.522} C_DIS
LIN {X -0.003,Y -482.174,Z 244.797,A 0.000,B 0.000,C 90.000,E1 359.484} C_DIS
LIN {X -0.175,Y -483.857,Z 244.782,A 0.000,B 0.000,C 90.000,E1 356.731} C_DIS
LIN {X 0.105,Y -485.496,Z 244.770,A 0.000,B 0.000,C 90.000,E1 354.546} C_DIS
LIN {X 0.100,Y -490.146,Z 244.748,A 0.000,B 0.000,C 90.000,E1 350.566} C_DIS
LIN {X -0.059,Y -493.581,Z 244.738,A 0.000,B 0.000,C 90.000,E1 348.757} C_DIS
LIN {X 0.099,Y -503.004,Z 244.717,A 0.000,B 0.000,C 90.000,E1 345.117} C_DIS
LIN {X 0.170,Y -507.112,Z 244.709,A 0.000,B 0.000,C 90.000,E1 343.614} C_DIS
LIN {X 0.139,Y -509.557,Z 244.704,A 0.000,B 0.000,C 90.000,E1 342.725} C_DIS
LIN {X -0.143,Y -513.716,Z 244.696,A 0.000,B 0.000,C 90.000,E1 341.275} C_DIS
LIN {X -0.123,Y -522.862,Z 244.680,A 0.000,B 0.000,C 90.000,E1 338.337} C_DIS
LIN {X -0.304,Y -528.820,Z 244.670,A 0.000,B 0.000,C 90.000,E1 336.613} C_DIS
LIN {X 0.063,Y -534.873,Z 244.660,A 0.000,B 0.000,C 90.000,E1 334.845} C_DIS
LIN {X -0.179,Y -542.158,Z 244.649,A 0.000,B 0.000,C 90.000,E1 332.871} C_DIS
LIN {X -0.237,Y -548.564,Z 244.640,A 0.000,B 0.000,C 90.000,E1 331.179} C_DIS
LIN {X 0.301,Y -552.779,Z 244.634,A 0.000,B 0.000,C 90.000,E1 329.999} C_DIS
LIN {X -0.277,Y -557.849,Z 244.626,A 0.000,B 0.000,C 90.000,E1 328.663} C_DIS
LIN {X 0.094,Y -566.994,Z 244.612,A 0.000,B 0.000,C 90.000,E1 326.135} C_DIS
LIN {X 0.189,Y -573.310,Z 244.603,A 0.000,B 0.000,C 90.000,E1 324.482} C_DIS
LIN {X -0.035,Y -577.402,Z 244.597,A 0.000,B 0.000,C 90.000,E1 323.417} C_DIS
LIN {X -0.020,Y -580.138,Z 244.592,A 0.000,B 0.000,C 90.000,E1 322.603} C_DIS
LIN {X 0.204,Y -585.527,Z 244.583,A 0.000,B 0.000,C 90.000,E1 320.964} C_DIS
LIN {X -0.312,Y -596.431,Z 244.567,A 0.000,B 0.000,C 90.000,E1 318.081} C_DIS
LIN {X 0.086,Y -600.475,Z 244.561,A 0.000,B 0.000,C 90.000,E1 316.986} C_DIS
LIN {X 0.343,Y -605.298,Z 244.554,A 0.000,B 0.000,C 90.000,E1 315.648} C_DIS
LIN {X 0.247,Y -609.499,Z 244.547,A 0.000,B 0.000,C 90.000,E1 314.352} C_DIS
LIN {X -0.298,Y -611.635,Z 244.542,A 0.000,B 0.000,C 90.000,E1 313.623} C_DIS
LIN {X 0.315,Y -614.143,Z 244.536,A 0.000,B 0.000,C 90.000,E1 312.528} C_DIS
LIN {X -0.028,Y -615.188,Z 244.534,A 0.000,B 0.000,C 90.000,E1 312.043} C_DIS
LIN {X 0.222,Y -617.046,Z 244.528,A 0.000,B 0.000,C 90.000,E1 310.987} C_DIS
LIN {X -0.206,Y -618.337,Z 244.524,A 0.000,B 0.000,C 90.000,E1 310.253} C_DIS
LIN {X -0.224,Y -619.530,Z 244.519,A 0.000,B 0.000,C 90.000,E1 309.483} C_DIS
LIN {X -0.305,Y -620.931,Z 244.514,A 0.000,B 0.000,C 90.000,E1 308.463} C_DIS
LIN {X 0.178,Y -621.874,Z 244.509,A 0.000,B 0.000,C 90.000,E1 307.649} C_DIS
LIN {X 0.292,Y -622.597,Z 244.505,A 0.000,B 0.000,C 90.000,E1 306.870} C_DIS
LIN {X -0.086,Y -623.072,Z 244.501,A 0.000,B 0.000,C 90.000,E1 306.137} C_DIS
LIN {X 0.011,Y -623.551,Z 244.495,A 0.000,B 0.000,C 90.000,E1 305.105} C_DIS
LIN {X 0.124,Y -623.726,Z 244.489,A 0.000,B 0.000,C 90.000,E1 304.072} C_DIS
LIN {X -0.279,Y -623.706,Z 244.484,A 0.000,B 0.000,C 90.000,E1 303.086} C_DIS
LIN {X 0.030,Y -623.263,Z 244.479,A 0.000,B 0.000,C 90.000,E1 302.291} C_DIS
LIN {X 0.123,Y -621.878,Z 244.472,A 0.000,B 0.000,C 90.000,E1 301.003} C_DIS
LIN {X -0.107,Y -621.165,Z 244.470,A 0.000,B 0.000,C 90.000,E1 300.512} C_DIS
LIN {X 0.157,Y -618.810,Z 244.462,A 0.000,B 0.000,C 90.000,E1 299.205} C_DIS
LIN {X 0.122,Y -617.152,Z 244.458,A 0.000,B 0.000,C 90.000,E1 298.437} C_DIS
LIN {X 0.321,Y -614.157,Z 244.451,A 0.000,B 0.000,C 90.000,E1 297.129} C_DIS
LIN {X 0.214,Y -611.495,Z 244.445,A 0.000,B 0.000,C 90.000,E1 296.104} C_DIS
LIN {X 0.025,Y -607.966,Z 244.438,A 0.000,B 0.000,C 90.000,E1 294.823} C_DIS
LIN {X -0.050,Y -603.157,Z 244.428,A 0.000,B 0.000,C 90.000,E1 293.003} C_DIS
LIN {X -0.221,Y -598.129,Z 244.416,A 0.000,B 0.000,C 90.000,E1 290.918} C_DIS
LIN {X 0.153,Y -593.928,Z 244.406,A 0.000,B 0.000,C 90.000,E1 289.033} C_DIS
LIN {X -0.218,Y -588.860,Z 244.393,A 0.000,B 0.000,C 90.000,E1 286.677} C_DIS
LIN {X -0.112,Y -585.779,Z 244.384,A 0.000,B 0.000,C 90.000,E1 285.064} C_DIS
LIN {X 0.242,Y -582.125,Z 244.372,A 0.000,B 0.000,C 90.000,E1 282.883} C_DIS
LIN {X -0.215,Y -578.057,Z 244.355,A 0.000,B 0.000,C 90.000,E1 279.962} C_DIS
LIN {X -0.078,Y -575.278,Z 244.340,A 0.000,B 0.000,C 90.000,E1 277.239} C_DIS
LIN {X 0.082,Y -573.642,Z 244.328,A 0.000,B 0.000,C 90.000,E1 275.049} C_DIS
LIN {X 0.247,Y -572.674,Z 244.296,A 0.000,B 0.000,C 90.000,E1 269.312} C_DIS
LIN {X -0.163,Y -576.390,Z 244.266,A 0.000,B 0.000,C 90.000,E1 263.913} C_DIS
LIN {X 0.273,Y -579.275,Z 244.253,A 0.000,B 0.000,C 90.000,E1 261.432} C_DIS
LIN {X 0.158,Y -582.246,Z 244.241,A 0.000,B 0.000,C 90.000,E1 259.285} C_DIS
LIN {X -0.047,Y -583.951,Z 244.235,A 0.000,B 0.000,C 90.000,E1 258.229} C_DIS
LIN {X -0.306,Y -586.452,Z 244.226,A 0.000,B 0.000,C 90.000,E1 256.645} C_DIS
LIN {X 0.261,Y -588.086,Z 244.220,A 0.000,B 0.000,C 90.000,E1 255.519} C_DIS
LIN {X 0.129,Y -589.705,Z 244.214,A 0.000,B 0.000,C 90.000,E1 254.464} C_DIS
LIN {X 0.023,Y -591.356,Z 244.206,A 0.000,B 0.000,C 90.000,E1 253.142} C_DIS
LIN {X 0.263,Y -592.253,Z 244.201,A 0.000,B 0.000,C 90.000,E1 252.054} C_DIS
LIN {X -0.236,Y -592.634,Z 244.195,A 0.000,B 0.000,C 90.000,E1 251.040} C_DIS
LIN {X 0.217,Y -592.798,Z 244.189,A 0.000,B 0.000,C 90.000,E1 249.934} C_DIS
LIN {X -0.086,Y -592.714,Z 244.183,A 0.000,B 0.000,C 90.000,E1 248.901} C_DIS
LIN {X -0.180,Y -592.062,Z 244.177,A 0.000,B 0.000,C 90.000,E1 247.847} C_DIS
LIN {X -0.070,Y -591.620,Z 244.174,A 0.000,B 0.000,C 90.000,E1 247.305} C_DIS
LIN {X -0.053,Y -589.984,Z 244.167,A 0.000,B 0.000,C 90.000,E1 245.973} C_DIS
LIN {X -0.083,Y -588.623,Z 244.162,A 0.000,B 0.000,C 90.000,E1 245.177} C_DIS
LIN {X -0.002,Y -586.516,Z 244.156,A 0.000,B 0.000,C 90.000,E1 244.101} C_DIS
LIN {X 0.308,Y -584.080,Z 244.150,A 0.000,B 0.000,C 90.000,E1 242.999} C_DIS
LIN {X -0.055,Y -580.716,Z 244.143,A 0.000,B 0.000,C 90.000,E1 241.691} C_DIS
LIN {X 0.179,Y -577.781,Z 244.137,A 0.000,B 0.000,C 90.000,E1 240.589} C_DIS
LIN {X -0.136,Y -574.632,Z 244.131,A 0.000,B 0.000,C 90.000,E1 239.537} C_DIS
LIN {X -0.374,Y -570.442,Z 244.123,A 0.000,B 0.000,C 90.000,E1 238.201} C_DIS
LIN {X 0.093,Y -565.949,Z 244.116,A 0.000,B 0.000,C 90.000,E1 236.786} C_DIS
LIN {X -0.174,Y -559.034,Z 244.103,A 0.000,B 0.000,C 90.000,E1 234.609} C_DIS
LIN {X -0.149,Y -555.539,Z 244.097,A 0.000,B 0.000,C 90.000,E1 233.497} C_DIS
LIN {X -0.101,Y -549.397,Z 244.086,A 0.000,B 0.000,C 90.000,E1 231.537} C_DIS
LIN {X 0.103,Y -544.086,Z 244.077,A 0.000,B 0.000,C 90.000,E1 229.828} C_DIS
LIN {X -0.223,Y -538.695,Z 244.067,A 0.000,B 0.000,C 90.000,E1 228.162} C_DIS
LIN {X 0.062,Y -533.278,Z 244.058,A 0.000,B 0.000,C 90.000,E1 226.419} C_DIS
LIN {X -0.105,Y -528.671,Z 244.050,A 0.000,B 0.000,C 90.000,E1 225.000} C_DIS
LIN {X -0.042,Y -523.113,Z 244.040,A 0.000,B 0.000,C 90.000,E1 223.257} C_DIS
LIN {X -0.171,Y -516.840,Z 244.029,A 0.000,B 0.000,C 90.000,E1 221.229} C_DIS
LIN {X -0.019,Y -510.696,Z 244.018,A 0.000,B 0.000,C 90.000,E1 219.152} C_DIS
LIN {X -0.135,Y -503.935,Z 244.004,A 0.000,B 0.000,C 90.000,E1 216.790} C_DIS
LIN {X -0.128,Y -497.959,Z 243.993,A 0.000,B 0.000,C 90.000,E1 214.692} C_DIS
LIN {X -0.129,Y -492.876,Z 243.983,A 0.000,B 0.000,C 90.000,E1 212.880} C_DIS
LIN {X 0.135,Y -487.187,Z 243.971,A 0.000,B 0.000,C 90.000,E1 210.718} C_DIS
LIN {X 0.179,Y -481.739,Z 243.959,A 0.000,B 0.000,C 90.000,E1 208.565} C_DIS
LIN {X 0.032,Y -475.485,Z 243.943,A 0.000,B 0.000,C 90.000,E1 205.796} C_DIS
LIN {X -0.223,Y -471.011,Z 243.931,A 0.000,B 0.000,C 90.000,E1 203.643} C_DIS
LIN {X 0.217,Y -464.303,Z 243.910,A 0.000,B 0.000,C 90.000,E1 199.812} C_DIS
LIN {X -0.020,Y -459.972,Z 243.894,A 0.000,B 0.000,C 90.000,E1 196.985} C_DIS
LIN {X 0.122,Y -455.743,Z 243.877,A 0.000,B 0.000,C 90.000,E1 193.772} C_DIS
LIN {X -0.034,Y -453.747,Z 243.868,A 0.000,B 0.000,C 90.000,E1 192.187} C_DIS
LIN {X -0.066,Y -450.724,Z 243.853,A 0.000,B 0.000,C 90.000,E1 189.613} C_DIS
LIN {X 0.086,Y -448.055,Z 243.839,A 0.000,B 0.000,C 90.000,E1 187.004} C_DIS
LIN {X -0.003,Y -445.782,Z 243.825,A 0.000,B 0.000,C 90.000,E1 184.416} C_DIS
LIN {X -0.033,Y -444.179,Z 243.814,A 0.000,B 0.000,C 90.000,E1 182.465} C_DIS
LIN {X 0.194,Y -443.036,Z 243.805,A 0.000,B 0.000,C 90.000,E1 180.802} C_DIS
LIN {X -0.123,Y -441.499,Z 243.790,A 0.000,B 0.000,C 90.000,E1 178.224} C_DIS
LIN {X -0.179,Y -440.503,Z 243.772,A 0.000,B 0.000,C 90.000,E1 174.951} C_DIS
LIN {X -0.035,Y -440.303,Z 243.752,A 0.000,B 0.000,C 90.000,E1 171.319} C_DIS
LIN {X -0.108,Y -440.822,Z 243.737,A 0.000,B 0.000,C 90.000,E1 168.701} C_DIS
LIN {X -0.025,Y -442.443,Z 243.715,A 0.000,B 0.000,C 90.000,E1 164.755} C_DIS
LIN {X 0.058,Y -443.756,Z 243.701,A 0.000,B 0.000,C 90.000,E1 162.127} C_DIS
LIN {X 0.036,Y -445.473,Z 243.686,A 0.000,B 0.000,C 90.000,E1 159.518} C_DIS
LIN {X 0.102,Y -447.552,Z 243.674,A 0.000,B 0.000,C 90.000,E1 157.230} C_DIS
LIN {X -0.131,Y -450.323,Z 243.659,A 0.000,B 0.000,C 90.000,E1 154.665} C_DIS
LIN {X -0.090,Y -453.640,Z 243.645,A 0.000,B 0.000,C 90.000,E1 152.076} C_DIS
LIN {X 0.068,Y -456.455,Z 243.634,A 0.000,B 0.000,C 90.000,E1 150.127} C_DIS
LIN {X -0.157,Y -459.963,Z 243.622,A 0.000,B 0.000,C 90.000,E1 147.916} C_DIS
LIN {X 0.082,Y -464.157,Z 243.608,A 0.000,B 0.000,C 90.000,E1 145.341} C_DIS
LIN {X -0.117,Y -466.739,Z 243.599,A 0.000,B 0.000,C 90.000,E1 143.783} C_DIS
LIN {X 0.248,Y -468.643,Z 243.592,A 0.000,B 0.000,C 90.000,E1 142.477} C_DIS
LIN {X -0.170,Y -471.307,Z 243.581,A 0.000,B 0.000,C 90.000,E1 140.642} C_DIS
LIN {X -0.098,Y -472.913,Z 243.574,A 0.000,B 0.000,C 90.000,E1 139.380} C_DIS
LIN {X 0.214,Y -473.959,Z 243.569,A 0.000,B 0.000,C 90.000,E1 138.405} C_DIS
LIN {X -0.042,Y -475.159,Z 243.562,A 0.000,B 0.000,C 90.000,E1 137.187} C_DIS
